(* CODESYS project SNDLTN_Domoticz.library
   Company: Sandolution
   Title: SNDLTN_Domoticz
   Description: Library to control Domoticz from a CoDeSys PLC using JSON over HTTP/MQTT.
   Author: S. Verbeek
   Version: 2.5.201026

Project tree, tasks and I/O mapping:
  libraries: StringUtils, * (System); Standard, * (System); CAA Real Time Clock Extern, * (CAA Technical Workgroup); SNDLTN_HTTP, 1.2.200929 (Sandolution); SNDLTN_MQTT, 1.2.200929 (Sandolution); SNDLTN_JSON, 1.2 (Sandolution)
  Constants/
    global variables Domoticz_Constants
    global variables Domoticz_Properties
  Enums/
    data type Domoticz_eErrors
    data type _Domoticz_eObjectDataType
    data type _Domoticz_eDataSource
    data type _Domoticz_eCommandType
    data type Domoticz_eSValues_Colors
    data type Domoticz_eHumidityStatus
    data type Domoticz_eForecast
    data type _Domoticz_eHTTP_PropertyNames
    data type Domoticz_eSValues_TempHumBaro
    data type Domoticz_eSValues_General
    data type Domoticz_eSValues_Wind
    data type Domoticz_eSValues_Rain
    data type Domoticz_eSValues_Usage
    data type Domoticz_eSValues_P1
    data type _Domoticz_eMQTT_PropertyNames
  Function Blocks/
    Objects/
      function block _Domoticz_ObjectBool_InOut [ST]: Main
      function block _Domoticz_ObjectReal_InOut [ST]: Main, rScalingSet
      function block _Domoticz_ObjectInt_InOut [ST]: Main, xUseOnlyNValue
      function block _Domoticz_Object [ST]: Main, ForceSet, RegisterSlave, xUpdateReceived, xDataTimedOut, sDeviceType, dtLastUpdate, eDataSource, eCommandType
      function block _Domoticz_ObjectString_InOut [ST]: Main
      function block _Domoticz_ObjectArrayReal_InOut [ST]: Main, arScalingSet
      function block _Domoticz_ObjectArrayReal_Out [ST]: Main, arScalingAct
      function block _Domoticz_ObjectBool_Out [ST]: Main
      function block _Domoticz_ObjectInt_Out [ST]: Main, iValueSetLimitLow, iValueSetLimitHigh
      function block _Domoticz_ObjectReal_Out [ST]: Main, rScalingAct
      function block _Domoticz_ObjectString_Out [ST]: Main
    Hardware/
      Weather/
        function block Domoticz_DarkSky [ST]: Main
        function block Domoticz_BuienAlarm [ST]: Main
        function block Domoticz_BuienRadar [ST]: Main
        function block Domoticz_OpenWeatherMap [ST]: Main
        function block Domoticz_WeatherBit [ST]: Main
        function block Domoticz_SunMoon [ST]: Main
        function block Domoticz_AccuWeather [ST]: Main
        function block Domoticz_BuienRadar_Forecast [ST]: Main
      Custom/
        function block Domoticz_CustomDimmer [ST]: Main, xUseOnlyNValue
        function block Domoticz_CustomSwitch [ST]: Main, xInvert
        function block Domoticz_CustomSensor [ST]: Main, rScalingSet, rScalingAct
        function block Domoticz_CustomString [ST]: Main
        function block Domoticz_CustomSensors [ST]: Main, arScalingSet, arScalingAct
      System/Network/
        function block Domoticz_SystemAliveChecker [ST]: Main
        function block Domoticz_MotherboardSensors [ST]: Main, rThresholdCPUHigh, rThresholdCPUMax, rThresholdMemoryHigh, rThresholdMemoryMax, rThresholdHDDHigh, rThresholdHDDMax, rThresholdTemperatureHigh, rThresholdTemperatureMax
        function block Domoticz_UPSMonitor [ST]: Main, rThresholdChargeLevelLow, rThresholdChargeLevelCritical, rThresholdLoadLevelHigh, rThresholdLoadLevelMax, rThresholdFrequency, rThresholdVoltage
        function block Domoticz_SpeedTest [ST]: Main, tThresholdPingHigh, rThresholdDownloadSpeedLow, rThresholdUploadSpeedLow
      Devices/
        function block Domoticz_MiFlora [ST]: Main, rThresholdMoistureLow, rThresholdFertilityLow
        function block Domoticz_HueLight [ST]: Main, tFadeTime, tFadeUpdateTime, xFading
        function block Domoticz_Tasmota [ST]: Main, rThresholdCurrentHigh, rThresholdCurrentMax, rThresholdPowerUsageHigh, rThresholdPowerUsageToday, rThresholdTemperatureHigh, rThresholdTemperatureLow, rThresholdHumidityHigh, rThresholdHumidityLow, rThresholdCarbonDioxideHigh, rThresholdCarbonDioxideCritical, rThresholdParticlesHigh_1um, rThresholdParticlesHigh_2_5um, rThresholdParticlesHigh_10um, rThresholdVoltage
        function block Domoticz_GoogleDevices [ST]: Main
        function block Domoticz_Life360 [ST]: Main, xArrivedHome, xLeftHome
        function block Domoticz_HueSensor [ST]: Main
        function block Domoticz_HuePlug [ST]: Main
        function block Domoticz_HueSwitch [ST]: Main
      Climate/Energy/
        function block Domoticz_NefitEasy [ST]: Main, rThresholdPressureLow, rThresholdGasUsageToday
        function block Domoticz_UsageMeter [ST]: Main, rThresholdUsageToday, sUnit
        function block Domoticz_P1Meter [ST]: Main, rThresholdGasUsageToday, rThresholdPowerUsageHigh, rThresholdPowerUsageToday, rThresholdVoltage
    Connector/
      function block _Domoticz_Connector_Out [ST]: Main, xDataTimeOut
      function block _Domoticz_Connector_InOut [ST]: tForceSetValues, Main, xForceSetValues
      function block _Domoticz_Connector [ST]: Main, sInstanceName
      function block _Domoticz_Connector_InOut_Extended [ST]: tDataTimeOut, Main
    Server/
      function block _Domoticz_Server [ST]: Main, udiUpdateRate_HTTP, HTTP_DataTwilight, MQTT_Main, HTTP_Main, MQTT_DataObject_In, MQTT_DataObject_Out, SystemTime, tSlaveErrorResetTime, Configure_AutoSyncClock, Configure_MQTT, Configure_HTTP, Configure_Twilight, xAutoReconnect, tDataForceSetValues, udiUpdateRate_MQTT, xStartUpDone, ErrorHandling, ascActiveSlaveErrors
      function block Domoticz_Server [ST]
      function block _Domoticz_Server_HTTP_Object [ST]: Main, ResetObjectData, DataObject_In
    Other/
      function block Domoticz_ServerLog [ST]: ShiftArray, Main
      function block Domoticz_ErrorInterface [ST]: Main, sErrorInfo, tErrorDelay
      function block _Domoticz_SwitchPoint [ST]: Main
  Functions/
    function _Domoticz_StringToReal [ST]
    function _Domoticz_StringToByte [ST]
    function _Domoticz_StringExtractColor [ST]
    function _Domoticz_RoundDecimals [ST]
    function _Domoticz_EqualWithWindow [ST]
    function _Domoticz_StringExtractAfterDot [ST]
    function _Domoticz_ColorFactor [ST]
  Structs/
    data type Domoticz_scObjectData
    data type Domoticz_scTwilightData
    data type Domoticz_scColorData
    data type Domoticz_scConnector
    data type Domoticz_scError
  Variables/
  Visualizations/
  text list GlobalTextList
  program ChangeLog [ST]
*)

// Enums/Domoticz_eErrors
{attribute 'qualified_only'}
{attribute 'to_string'}
TYPE Domoticz_eErrors:
(
	NoError 								:= 0,		// No error
	                                		
	//0-99 :SERVER                 		
	ServerStarting							:= 1,		//First data refresh cycle (HTTP) active
	HTTPConnectionLost						:= 10,		//Lost connection with HTTP broker
	HTTPUpdateTimeOut						:= 11,		//Timeout on last update
	MQTTConnectionLost						:= 20,		//Lost connection with MQTT broker
	MQTTUpdateTimeOut						:= 21,		//Timeout on last update
	ErrorHandlerArrayFull					:= 30,		//Array full
	ErrorHandlerEntryNotFound				:= 31,		//Entry not found in array
                                    		
	//100-199 :OBJECTS             		
	ObjectMaxReached						:= 100, 	//Maximal amount of slaves connected
	ObjectRegistrationNotPossible			:= 101,		//Register slave not possible
	ObjectInvalidData						:= 102,		//Failed during reading of HTTP data
	ObjectDataTimeOut						:= 103,		//TimeOut of received data
	                                		
	//200-999 :HARDWARE            		
	                                		
	//200-249 :Motherboard         		
	Motherboard_CpuUsageHigh				:= 210,		//Motherboard high CPU usage (>75%)
	Motherboard_CpuUsageMax					:= 211,		//Motherboard high CPU usage (>95%)
	Motherboard_MemoryUsageHigh				:= 220,		//Motherboard high memory usage (>75%)
	Motherboard_MemoryUsageMax				:= 221,		//Motherboard high memory usage (>95%)
	Motherboard_HddUsageHigh				:= 230,		//Motherboard high HDD usage (>75%)
	Motherboard_HddUsageMax					:= 231,		//Motherboard high HDD usage (>90%)
	Motherboard_TemperatureHigh				:= 240,		//Motherboard high temperature (> C60)
	Motherboard_TemperatureMax				:= 241,		//Motherboard high temperature (> C80)
	//250-299 :Speedtest           		
	SpeedTest_PingHigh						:= 260,		//Speedtest high ping
	SpeedTest_DownloadSpeedLow				:= 270,		//Speedtest download speed low
	SpeedTest_UploadSpeedLow				:= 271,		//Speedtest upload speed low                            
	//300-349 :MiFlora             		      
	MiFlora_MoistureLow						:= 310,		//MiFlora low moisture (< 25%)
	MiFlora_FertilityLow					:= 311,		//MiFlora low fertility (< 500uS/cm)
	//350-399 :Tasmota   
	Tasmota_PowerFailure					:= 350,		//Tasmota Mains voltage lost
	Tasmota_PowerUsageToday					:= 351,		//Tasmota high power usage (today)
	Tasmota_PowerUsageHigh					:= 352,		//Tasmota high actual power usage
	Tasmota_CurrentHigh						:= 355,		//Tasmota Load level at high level
	Tasmota_CurrentMax						:= 356,		//Tasmota Load level at max level        		
	Tasmota_TemperatureHigh					:= 360,		//Tasmota temperature too high
	Tasmota_TemperatureLow					:= 361,		//Tasmota temperature too low
	Tasmota_HumidityHigh					:= 365,		//Tasmota humidity too high
	Tasmota_HumidityLow						:= 366,		//Tasmota humidity too low
	Tasmota_CarbonDioxideHigh				:= 370,		//Tasmota carbondioxide high
	Tasmota_CarbonDioxideCritical			:= 371,		//Tasmota carbondioxide critical
	Tasmota_ParticlesHigh_1um				:= 380,		//Tasmota carbondioxide high PM1
	Tasmota_ParticlesHigh_2_5um				:= 381,		//Tasmota carbondioxide high PM2.5
	Tasmota_ParticlesHigh_10um				:= 382,		//Tasmota carbondioxide high PM10
	//400-449 :NefitEasy
	Nefit_PressureLow						:= 410,		//Nefit low pressure
	Nefit_GasUsageToday						:= 420,		//Nefit high gas usage (today)
	//450-499 :UsageMeter          		
	UsageMeter_UsageToday					:= 460,		//UsageMeter high usage (today)
	//500-549 :P1 Meter            		
	P1_PowerFailure							:= 510,		//P1Meter Mains voltage lost
	P1_PowerUsageToday						:= 520,		//P1Meter high power usage (today)
	P1_PowerUsageHigh						:= 521,		//P1Meter high actual power usage
	P1_GasUsageToday						:= 530,		//P1Meter high gas usage (today)
	//550-599 :UPS                 		
	UPS_PowerFailure						:= 560,		//UPS Mains voltage lost
	UPS_ChargeLevelLow						:= 570,		//UPS Capacity at warning level (<50%)
	UPS_ChargeLevelCritical					:= 571,		//UPS Capacity at critical level (<25%)
	UPS_LoadLevelHigh						:= 580,		//UPS Load level at high level (>75%)
	UPS_LoadLevelMax						:= 581,		//UPS Load level at critical level (>95%)
	UPS_BackupTime_5Min						:= 590,		//UPS Backup time (<5 min)
	UPS_BackupTime_1Min						:= 591,		//UPS Backup time (<1 min)
	//600-649
	Life360_LeftHome						:= 600,		//Life 360 left home
	Life360_ArrivedHome						:= 601,		//Life 360 arrived home
	//650-699                       		
	//700-749                       		
	//750-799                       		
	//800-849                       		
	//850-899                       		
	//900-999 :CUSTOM              		
	//Doors/Windows
	Custom_DoorOpened						:= 910,
	Custom_DoorClosed						:= 911,
	Custom_WindowOpened						:= 915,
	Custom_WindowClosed						:= 916,
	               
	//Safety     
	Custom_AlarmArmed_Stay					:= 920,
	Custom_AlarmArmed_Away					:= 921,
	Custom_AlarmDisarmed					:= 922,            		
	Custom_MovementDetected					:= 925,	
	
	//Temperature                        		  
	Custom_TemperatureHigh					:= 930,
	Custom_TemperatureLow					:= 931,
	Custom_TemperatureOutOfRange			:= 932,
	
	//Humidity                        		  
	Custom_HumidityHigh						:= 935,
	Custom_HumidityLow						:= 936,
	Custom_HumidityOutOfRange				:= 937,
	
	//Weather
	Custom_RainExpected						:= 940,
	Custom_SnowExpected						:= 941,
	Custom_FrostExpected					:= 942,
	
	//Power                   		      
	Custom_PowerFailure						:= 950,
	Custom_PowerUsageHigh					:= 951,
	Custom_PowerUsageToday					:= 952,
	         
	//System                       		
	Custom_RetainDataInvalid				:= 960,
	
	//Network
	Custom_HostUnreachable					:= 965,
	Custom_HostUnknown						:= 966,

	//Devices                               		
	Custom_ProgramComplete					:= 970,
	Custom_Triggered						:= 971,
	Custom_Activated						:= 975,
	Custom_Active							:= 976,
	Custom_Deactivated						:= 977,
	Custom_Inactive							:= 978,
	
	//Other
	Custom_Spare0							:= 990,
	Custom_Spare1							:= 991,
	Custom_Spare2							:= 992,
	Custom_Spare3							:= 993,
	Custom_Spare4							:= 994,
	Custom_Spare5							:= 995,
	Custom_Spare6							:= 996,
	Custom_Spare7							:= 997,
	Custom_Spare8							:= 998,
	Custom_Spare9							:= 999,
	
		
	//1000-1999 :HTTP ERRORS (SEE LIBRARY SNDLTN_HTTP)
	HTTP_MissingPostValue					:= 1001, 	//Current request type needs a post value
	HTTP_ParsingError						:= 1002, 	//Error while parsing the response
	HTTP_InvalidIdentifier					:= 1003,	//Invalid identifier (probably 0)
	
	//NBS errors (ported from 6001-6099)
	HTTP_NBS_TimeOut 						:= 1100,	//Time limit exceeded
	HTTP_NBS_InvalidAddress					:= 1101,	//Address invalid
	HTTP_NBS_InvalidHandle					:= 1102,	//Handle invalid
	HTTP_NBS_InvalidPointer					:= 1103,	//Data pointer invalid
	HTTP_NBS_InvalidSize					:= 1104,	//Data size invalid
	HTTP_NBS_ReceiveUDP						:= 1105,	//Error receiving data via UDP
	HTTP_NBS_SendUDP						:= 1106,	//Error sending data via UDP
	HTTP_NBS_SentIncompleteUDP				:= 1107,	//Not all data is sent.
	HTTP_NBS_OpenUDP						:= 1108,	//Couldn't open UDP connection
	HTTP_NBS_CloseUDP						:= 1109,	//Couldn't close UDP connection
	HTTP_NBS_SendTCP						:= 1110,	//Error sending data via TCP
	HTTP_NBS_ReceiveTCP						:= 1111,	//Error receiving data via TCP
	HTTP_NBS_OpenTCP						:= 1112,	//Couldn't open TCP connection
	HTTP_NBS_ConnectTCP						:= 1113,	//Couldn't connect TCP connection
	HTTP_NBS_CloseTCP						:= 1114,	//Couldn't close TCP connection
	HTTP_NBS_ServerTCP						:= 1115,	//Server error TCP
	HTTP_NBS_WrongParameter					:= 1116,	//Wrong parameters entered
	HTTP_NBS_Unknown						:= 1117,	//Not specified
	
	
	//2000-2999 :MQTT ERRORS (SEE LIBRARY SNDLTN_MQTT)
	
	//Custom errors
	MQTT_InvalidMQTT						:= 2000,	//Invalid MQTT response
	MQTT_BufferOverflow						:= 2001,	//Overflow from method
	MQTT_ConnectionLost						:= 2002,	//Connection with server lost
                                    		
	//Broker responses              		
	MQTT_RefusedProtocolVersion				:= 2010,	//Wrong protocol version
	MQTT_RefusedIdentifier					:= 2011,	//Identifier rejected
	MQTT_RefusedUserPass					:= 2012,	//Server unavailable
	MQTT_RefusedAuthorization				:= 2013,	//Authorization failed
	MQTT_ServerUnavailable					:= 2014,	//Server not available
		
	//NBS errors (ported from 6001-6099)
	MQTT_NBS_TimeOut 						:= 2100,	//Time limit exceeded
	MQTT_NBS_InvalidAddress					:= 2101,	//Address invalid
	MQTT_NBS_InvalidHandle					:= 2102,	//Handle invalid
	MQTT_NBS_InvalidPointer					:= 2103,	//Data pointer invalid
	MQTT_NBS_InvalidSize					:= 2104,	//Data size invalid
	MQTT_NBS_ReceiveUDP						:= 2105,	//Error receiving data via UDP
	MQTT_NBS_SendUDP						:= 2106,	//Error sending data via UDP
	MQTT_NBS_SentIncompleteUDP				:= 2107,	//Not all data is sent.
	MQTT_NBS_OpenUDP						:= 2108,	//Couldn't open UDP connection
	MQTT_NBS_CloseUDP						:= 2109,	//Couldn't close UDP connection
	MQTT_NBS_SendTCP						:= 2110,	//Error sending data via TCP
	MQTT_NBS_ReceiveTCP						:= 2111,	//Error receiving data via TCP
	MQTT_NBS_OpenTCP						:= 2112,	//Couldn't open TCP connection
	MQTT_NBS_ConnectTCP						:= 2113,	//Couldn't connect TCP connection
	MQTT_NBS_CloseTCP						:= 2114,	//Couldn't close TCP connection
	MQTT_NBS_ServerTCP						:= 2115,	//Server error TCP
	MQTT_NBS_WrongParameter					:= 2116,	//Wrong parameters entered
	MQTT_NBS_Unknown						:= 2117,	//Not specified
		
	//3000-3999 :JSON ERRORS (SEE LIBRARY SNDLTN_JSON)
	JSON_PropertiesArrayToSmall 			:= 3000,	//JSON Parser output array to small
	JSON_PropertySizeToSmall 				:= 3001		//JSON Size to small
);
END_TYPE

// Enums/_Domoticz_eObjectDataType
{attribute 'qualified_only'}
{attribute 'strict'}
{attribute 'conditionalshow'}
{attribute 'to_string'}
TYPE _Domoticz_eObjectDataType :
(
	NotUsed := 0,
	Identifier,
	Name,
	nValue,
	sValue1,
	sValue2,
	sValue3,
	sValue4,
	sValue5,
	sValue6,
	Color
);
END_TYPE

// Structs/Domoticz_scObjectData
TYPE Domoticz_scObjectData :
STRUCT
	//General
	uiIdentifier	:UINT;													//Identifier
	                  
	dtLastUpdate	:DATE_AND_TIME;											//Value latest updated
	dtTimeStamp		:DATE_AND_TIME;											//Latest read update
	                  
	asValue			:ARRAY[1..Domoticz_Constants.uiMaxSValues] OF STRING(JSON_Properties.uiJSONMaxPropertySize);	//Contains value if string
	iValue			:INT;													//Contains value if number
	
	//Indicate source of data
	eSource			:_Domoticz_eDataSource;									//1=MQTT 2=HTTP
	
	//Type of command (outgoing data)
	{attribute 'conditionalshow'}
	eCommand		:_Domoticz_eCommandType;								//Type of command to send
	
	{attribute 'conditionalshow'}
	sDeviceType		:STRING(Domoticz_Constants.uiObjectData_Type);			//Type of device

END_STRUCT
END_TYPE

// Structs/Domoticz_scTwilightData
TYPE Domoticz_scTwilightData :
STRUCT
	//Time
	dtSystem				:DATE_AND_TIME;
	todSystem				:TIME_OF_DAY;	
	dtServer				:DATE_AND_TIME;			//Server time is only retreived at twilight update interval
                              
	axHours					:ARRAY[0..23] OF BOOL;
                              
	xAstronomicRise			:BOOL;
	todAstronomicRise		:TIME_OF_DAY;
	                          
	xNauticRise				:BOOL;
	todNauticRise			:TIME_OF_DAY;
		                      
	xCivilRise				:BOOL;
	todCivilRise			:TIME_OF_DAY;
	                          
	xPreSunRise				:BOOL;
	todPreSunRise			:TIME_OF_DAY;
	xSunRise				:BOOL;
	todSunRise				:TIME_OF_DAY;
	xPostSunRise			:BOOL;
	todPostSunRise			:TIME_OF_DAY;
                              
	xSunAtSouth				:BOOL;
	todSunAtSouth			:TIME_OF_DAY;
	                          
	xPreSunSet				:BOOL;
	todPreSunSet			:TIME_OF_DAY;
	xSunSet					:BOOL;
	todSunSet				:TIME_OF_DAY;
	xPostSunSet				:BOOL;
	todPostSunSet			:TIME_OF_DAY;	
	                          
	xCivilSet				:BOOL;
	todCivilSet				:TIME_OF_DAY;	
	                          
	xNauticSet				:BOOL;
	todNauticSet			:TIME_OF_DAY;	
	                          
	xAstronomicSet			:BOOL;
	todAstronomicSet		:TIME_OF_DAY;
	                          
	todDayLength			:TIME_OF_DAY;
END_STRUCT
END_TYPE

// Enums/_Domoticz_eDataSource
{attribute 'qualified_only'}
{attribute 'strict'}
{attribute 'conditionalshow'} 
{attribute 'to_string'}
TYPE _Domoticz_eDataSource :
(
	All := 0,			//Allow all data sources
	MQTT,
	HTTP,
	PLC
);
END_TYPE

// Enums/_Domoticz_eCommandType
{attribute 'qualified_only'}
{attribute 'strict'}
{attribute 'conditionalshow'}
{attribute 'to_string'}
TYPE _Domoticz_eCommandType :
(
	Default := 0,
	SwitchLight,
	SwitchScene,
	SetColor,
	SetBrightness
);
END_TYPE

// Structs/Domoticz_scColorData
TYPE Domoticz_scColorData :
STRUCT
	byBrightness	:BYTE := 255;
	byRed			:BYTE;
	byGreen			:BYTE;
	byBlue			:BYTE;
	byColdWhite		:BYTE;
	byWarmWhite		:BYTE;
END_STRUCT
END_TYPE

// Enums/Domoticz_eSValues_Colors
{attribute 'qualified_only'}
{attribute 'strict'}
{attribute 'conditionalshow'}
{attribute 'to_string'}
TYPE Domoticz_eSValues_Colors :
(
	//Same order is also used in Constants.asProperty_Colors
	Brightness := 1,
	Red,
	Green,
	Blue,
	ColdWhite,
	WarmWhite
);
END_TYPE

// Structs/Domoticz_scConnector
TYPE Domoticz_scConnector :
STRUCT
	
	//Server status
	xServerConnected		:BOOL;						//Enabled and connected over HTTP and MQTT
	
	scTwilightData			:Domoticz_scTwilightData;	//Twilight data containing pulses also
	
	//Connected slave identifiers
	{attribute 'conditionalshow'}
	auiSlaveIdentifier		:ARRAY[1..Domoticz_Properties.uiMaxConnectedSlaves] OF UINT;

	uiSlaveTotal			:UINT;
	
	//Connected slave errors
	scSlaveError			:Domoticz_scError;
	
	//Forcing parameter
	tDataForceSetValues		:TIME := T#5S;				//Force set value if act is different
	
	//Input send data
	{attribute 'conditionalshow'}
	xNewObject_Tx			:BOOL;						//New values in object data
	{attribute 'conditionalshow'}
	scObjectData_Tx			:Domoticz_scObjectData;		//Object data
	
	//Output received data
	{attribute 'conditionalshow'}
	xNewObject_Rx			:BOOL;						//New values in object data
	{attribute 'conditionalshow'}
	scObjectData_Rx			:Domoticz_scObjectData;		//Object data
		
END_STRUCT
END_TYPE

// Enums/Domoticz_eHumidityStatus
{attribute 'qualified_only'}
{attribute 'to_string'} 
TYPE Domoticz_eHumidityStatus :
(
	Normal := 0,
	Comfortable := 1,
	Dry := 2,
	Wet := 3
);
END_TYPE

// Enums/Domoticz_eForecast
{attribute 'qualified_only'}
{attribute 'to_string'} 
TYPE Domoticz_eForecast :
(
	Stable := 0,
	Sunny := 1,
	PartlyCloudy := 2,
	Cloudy := 3,
	Rain := 4,
	Unknown := 5
);
END_TYPE

// Enums/_Domoticz_eHTTP_PropertyNames
{attribute 'qualified_only'}
{attribute 'strict'}
TYPE _Domoticz_eHTTP_PropertyNames :
(
	//General
	ObjectType := 1,
	Data,
	SwitchType,
	LastUpdate,
	//Switch
	Level,
	//Temp/Hum/Baro
	Temperature,
	DewPoint,
	Humidity,
	HumidityStatus,
	Barometer,
	Forecast,
	//Wind
	Speed,
	Chill,
	Gust,
	Direction,
	//Rain
	Rain,
	RainRate,
	//RGB(W)(W)
	Color,
	//Energy
	Counter,
	CounterToday,
	CounterDelivery,
	CounterDeliveryToday,
	Usage,
	UsageDelivery
);
END_TYPE

// Enums/Domoticz_eSValues_TempHumBaro
{attribute 'qualified_only'}
{attribute 'strict'}
{attribute 'conditionalshow'}
{attribute 'to_string'}
TYPE Domoticz_eSValues_TempHumBaro :
(
	//Same order is also used in Constants.asProperty_Colors
	Temperature := 1,
	Humidity,
	HumidityStatus,
	Barometer,
	Forecast,
	DewPoint
);
END_TYPE

// Enums/Domoticz_eSValues_General
{attribute 'qualified_only'}
{attribute 'strict'}
{attribute 'conditionalshow'}
{attribute 'to_string'}
TYPE Domoticz_eSValues_General :
(
	//Same order is also used in Constants.asProperty_Colors
	General := 1
);
END_TYPE

// Enums/Domoticz_eSValues_Wind
{attribute 'qualified_only'}
{attribute 'strict'}
{attribute 'conditionalshow'}
{attribute 'to_string'}
TYPE Domoticz_eSValues_Wind :
(
	//Same order is also used in Constants.asProperty_Colors
	Bearing := 1,
	Direction,
	Speed,
	Gust,
	Temperature,
	Chill
);
END_TYPE

// Enums/Domoticz_eSValues_Rain
{attribute 'qualified_only'}
{attribute 'strict'}
{attribute 'conditionalshow'}
{attribute 'to_string'}
TYPE Domoticz_eSValues_Rain :
(
	//Same order is also used in Constants.asProperty_Colors
	Rain := 1,
	RainRate
);
END_TYPE

// Enums/Domoticz_eSValues_Usage
{attribute 'qualified_only'}
{attribute 'strict'}
{attribute 'conditionalshow'}
{attribute 'to_string'}
TYPE Domoticz_eSValues_Usage :
(
	//Same order is also used in Constants.asProperty_Colors
	Usage := 1,
	UsageCumulative,	
	UsageToday 				//Additional from HTTP, not send by MQTT
);
END_TYPE

// Enums/Domoticz_eSValues_P1
{attribute 'qualified_only'}
{attribute 'strict'}
{attribute 'conditionalshow'}
{attribute 'to_string'}
TYPE Domoticz_eSValues_P1 :
(
	//Same order is also used in Constants.asProperty_Colors
	Usage1Cumulative := 1,
	Usage2Cumulative,
	Return1Cumulative,
	Return2Cumulative,
	UsageActual,
	ReturnActual,
	UsageToday,		//Additional from HTTP, not send by MQTT
	ReturnToday		//Additional from HTTP, not send by MQTT
);
END_TYPE

// Enums/_Domoticz_eMQTT_PropertyNames
{attribute 'qualified_only'}
{attribute 'strict'}
TYPE _Domoticz_eMQTT_PropertyNames :
(
	//General
	Identifier := 1,
	ObjectType,
	SwitchType,
	NValue,
	SValue1,
	SValue2,
	SValue3,
	SValue4,
	SValue5,
	SValue6,
	ColorR,
	ColorG,
	ColorB,
	ColorCW,
	ColorWW
);
END_TYPE

// Structs/Domoticz_scError
TYPE Domoticz_scError :
STRUCT
	xError				:BOOL := FALSE;
	eErrorID			:Domoticz_eErrors := Domoticz_eErrors.NoError;
	sErrorInstance		:STRING(Domoticz_Constants.uiInstanceName) := '';		//Contains instance name
	sErrorInfo			:STRING(Domoticz_Constants.uiErrorInfoSize) := '';		//Additional error info text
	udiUniqueID			:UDINT := 0;
END_STRUCT
END_TYPE

// Constants/Domoticz_Constants
{attribute 'qualified_only'}
{attribute 'conditionalshow'}
VAR_GLOBAL CONSTANT
	
	//**************************************************************************General
	uiObjectData_Type						:UINT			:= 32;		//Size of string
	uiInstanceName							:UINT			:= 128;		//Size of string
	uiMaxSValues							:UINT 			:= 8;		//Maximal S-values received, also change Domoticz_eObjectDataType and MQTT_In and HTTP_In
	uiMaxSValueSize							:UINT			:= 128;		//Maximal size of element

	uiErrorInfoSize							:UINT			:= 254;		//Size of additional error info text
	
	//**************************************************************************Types
	sType_Lighting1							:STRING(10)		:= 'Lighting 1';
	sType_Lighting2							:STRING(10)		:= 'Lighting 2';
	sType_Lighting3							:STRING(10)		:= 'Lighting 3';
	sType_Lighting4							:STRING(10)		:= 'Lighting 4';
	sType_Lighting5							:STRING(10)		:= 'Lighting 5';
	sType_LightSwitch						:STRING(12)		:= 'Light/Switch';
	sType_Security							:STRING(8)		:= 'Security';
	sSwitchType_Selector					:STRING(8)		:= 'Selector';
	sSwitchType_SelectorSwitch				:STRING(15)		:= 'Selector Switch';
	sSwitchType_Dimmer						:STRING(6)		:= 'Dimmer';
	sType_ColorSwitch						:STRING(12)		:= 'Color Switch';
	sType_TemperatureHumidityBaro			:STRING(22)		:= 'Temp + Humidity + Baro';
	sType_TemperatureHumidity				:STRING(15)		:= 'Temp + Humidity';
	sType_TemperatureBaro					:STRING(11)		:= 'Temp + Baro';
	sType_Temperature						:STRING(4)		:= 'Temp';
	sType_Humidity							:STRING(8)		:= 'Humidity';
	sType_AirQuality						:STRING(11)		:= 'Air Quality';
	sType_Wind								:STRING(4)		:= 'Wind';
	sType_Rain								:STRING(4)		:= 'Rain';
	sType_P1SmartMeter						:STRING(14)		:= 'P1 Smart Meter';
	sType_General							:STRING(7)		:= 'General';
	sType_kWh								:STRING(3)		:= 'kWh';
	sType_Energy							:STRING(6)		:= 'Energy';
	sType_Gas								:STRING(3)		:= 'Gas';
	
	//**************************************************************************Data
	sData_On								:STRING(2)		:= 'On';
	sData_Off								:STRING(3)		:= 'Off';
	sData_Open								:STRING(4)		:= 'Open';
	sData_Closed							:STRING(6)		:= 'Closed';
	sData_Locked							:STRING(6)		:= 'Locked';
	sData_Unlocked							:STRING(8)		:= 'Unlocked';
	sData_Normal							:STRING(6)		:= 'Normal';
	sData_Panic								:STRING(5)		:= 'Panic';
	
	//**************************************************************************MQTT
	//Below is present in MQTT data    
	//sPropertyMQTT_Battery					:STRING(7)		:= 'Battery';
	//sPropertyMQTT_RSSI					:STRING(4)		:= 'RSSI';
	//sPropertyMQTT_Description				:STRING(1)		:= 'description';
	sPropertyMQTT_DType						:STRING(5)		:= 'dtype';
	//sPropertyMQTT_ID						:STRING(2)		:= 'id';
	sPropertyMQTT_idx						:STRING(3)		:= 'idx';
	//sPropertyMQTT_Name					:STRING(4)		:= 'name';
	sPropertyMQTT_NValue					:STRING(6)		:= 'nvalue';
	sPropertyMQTT_SType						:STRING(5)		:= 'stype';
	sPropertyMQTT_SValue1					:STRING(7)		:= 'svalue1';
	sPropertyMQTT_SValue2					:STRING(7)		:= 'svalue2';
	sPropertyMQTT_SValue3					:STRING(7)		:= 'svalue3';
	sPropertyMQTT_SValue4					:STRING(7)		:= 'svalue4';
	sPropertyMQTT_SValue5					:STRING(7)		:= 'svalue5';
	sPropertyMQTT_SValue6					:STRING(7)		:= 'svalue6';
	//sPropertyMQTT_Unit					:STRING(4)		:= 'unit';
	//sPropertyMQTT_Color					:STRING(5)		:= 'Color';	
	
	//Commands 
	sCommandMQTT_uDevice					:STRING(19)		:= '"command":"udevice"';
	sCommandMQTT_SwitchLight				:STRING(23)		:= '"command":"switchlight"';	
	sCommandMQTT_SwitchScene				:STRING(23)		:= '"command":"switchscene"';	
	sCommandMQTT_Color						:STRING(33)		:= '"command":"setcolbrightnessvalue"';
	sCommandMQTT_Color_Value				:STRING(8)		:= '"color":';
	sCommandMQTT_Color_Mode					:STRING(1)		:= 'm';
	sCommandMQTT_Color_Temperature			:STRING(1)		:= 't';
	//Color command is defined at asProperty_Colors
	sCommandMQTT_idx						:STRING(6)		:= '"idx":';
	sCommandMQTT_sValues					:STRING(10)		:= '"svalue":"';
	sCommandMQTT_nValue						:STRING(9)		:= '"nvalue":';
	sCommandMQTT_SwitchOn					:STRING(16)		:= '"switchcmd":"On"';
	sCommandMQTT_SwitchOff					:STRING(17)		:= '"switchcmd":"Off"';
	sCommandMQTT_SwitchLevel				:STRING(23)		:= '"switchcmd":"Set Level"';
	sCommandMQTT_Level						:STRING(8)		:= '"level":';
	sCommandMQTT_Brightness					:STRING(13)		:= '"brightness":';
	
	//**************************************************************************HTTP
	sURL_HTTP								:STRING(7)		:= 'http://';	
	sURL_Twilight							:STRING(42)		:= '/json.htm?type=command&param=getSunRiseSet';
	sURL_Object								:STRING(27)		:= '/json.htm?type=devices&rid=';
	
	//Object
	sPropertyHTTP_Data						:STRING(4)		:= 'Data';
	sPropertyHTTP_Type						:STRING(4)		:= 'Type';
	sPropertyHTTP_SwitchType				:STRING(10)		:= 'SwitchType';
	sPropertyHTTP_LastUpdate				:STRING(10)		:= 'LastUpdate';
	
	//Temp/hum/baro
	sPropertyHTTP_Barometer					:STRING(9)		:= 'Barometer';
	sPropertyHTTP_Forecast					:STRING(8)		:= 'Forecast';
	sPropertyHTTP_DewPoint					:STRING(8)		:= 'DewPoint';
	sPropertyHTTP_Humidity					:STRING(8)		:= 'Humidity';
	sPropertyHTTP_HumidityStatus			:STRING(14)		:= 'HumidityStatus';
	sPropertyHTTP_Temperature				:STRING(4)		:= 'Temp';
	
	//Wind
	sPropertyHTTP_Direction					:STRING(9)		:= 'Direction';
	sPropertyHTTP_Chill						:STRING(5)		:= 'Chill';
	sPropertyHTTP_Gust						:STRING(4)		:= 'Gust';
	sPropertyHTTP_Speed						:STRING(5)		:= 'Speed';
	
	//Rain
	sPropertyHTTP_Rain						:STRING(4)		:= 'Rain';
	sPropertyHTTP_RainRate					:STRING(8)		:= 'RainRate';
	
	//RGB(W)(W)
	sPropertyHTTP_Color						:STRING(5)		:= 'Color';
	sPropertyHTTP_Level						:STRING(5)		:= 'Level';
	
	//Energy
	sPropertyHTTP_Counter					:STRING(7)		:= 'Counter';
	sPropertyHTTP_CounterToday				:STRING(12)		:= 'CounterToday';
	sPropertyHTTP_CounterDelivery			:STRING(12)		:= 'CounterDeliv';
	sPropertyHTTP_CounterDeliveryToday		:STRING(17)		:= 'CounterDelivToday';
	sPropertyHTTP_Usage						:STRING(5)		:= 'Usage';
	sPropertyHTTP_UsageDelivery				:STRING(10)		:= 'UsageDeliv';
	
	                            		
	//Twilight data                           		
	sPropertyHTTP_AstronomicRise			:STRING(17)		:= 'AstrTwilightStart';
	sPropertyHTTP_AstronomicSet				:STRING(15)		:= 'AstrTwilightEnd';
	sPropertyHTTP_CivilRise					:STRING(16)		:= 'CivTwilightStart';
	sPropertyHTTP_CivilSet					:STRING(14)		:= 'CivTwilightEnd';
	sPropertyHTTP_NauticRise				:STRING(17)		:= 'NautTwilightStart';
	sPropertyHTTP_NauticSet					:STRING(15)		:= 'NautTwilightEnd';
	sPropertyHTTP_SunRise					:STRING(7)		:= 'Sunrise';
	sPropertyHTTP_SunSet					:STRING(6)		:= 'Sunset';             		    	
	sPropertyHTTP_DayLength					:STRING(9)		:= 'DayLength';
	sPropertyHTTP_AtSouth					:STRING(10)		:= 'SunAtSouth';                            		
	sPropertyHTTP_SystemTime				:STRING(10)		:= 'ServerTime';
	
	
	//**************************************************************************COLOR
	uiProperty_ColorArraySize				:UINT := 6;
	asProperty_Colors						:ARRAY[1..uiProperty_ColorArraySize] OF STRING(2) := ['','r','g','b','cw','ww'];		//This order is also used in the array of sValues (2-6), 1 is brightness

END_VAR

// Constants/Domoticz_Properties
{attribute 'qualified_only'}
{attribute 'strict'}
VAR_GLOBAL CONSTANT
	//**************************************************************************General
	
	uiMaxConnectedSlaves					:UINT 	:= 256;			//Max connected slaves
	uiMaxHTTPConnections					:UINT 	:= 8;			//Max simultaneously connections
	uiHTTPStartUpCycles						:UINT 	:= 2;			//Number of cycles for HTTP to cycle before server reports connected
	
	uiActiveErrors							:UINT 	:= 32;			//Array size of active errors
	
	uiInterfaceLog_MaxEntries				:UINT 	:= 32;			//Maximal entries in log
	
	//MQTT Topics of Domoticz
	sMQTT_TopicReceive						:STRING(MQTT_Properties.uiMQTTMaxTopicSize) := 'domoticz/out';		//Out topic
	sMQTT_TopicSend							:STRING(MQTT_Properties.uiMQTTMaxTopicSize) := 'domoticz/in';		//In topic
	
END_VAR

// Function Blocks/Hardware/Climate/Energy/Domoticz_NefitEasy
{attribute 'conditionalshow_all_locals'}
FUNCTION_BLOCK Domoticz_NefitEasy EXTENDS _Domoticz_Connector_InOut
VAR_INPUT
	uiIdentifier_TemperatureSetpoint	:UINT;		//Setpoint temperature
	rTemperatureSetpoint_Set			:REAL;		//Setpoint temperature
	uiIdentifier_TemperatureRoom		:UINT;		//Actual temperature
	uiIdentifier_TemperatureFlow		:UINT;		//Flow temperature
	uiIdentifier_TemperatureOutside		:UINT;		//Outside temperature
	uiIdentifier_Pressure				:UINT;		//Heating pressure
	uiIdentifier_GasUsage				:UINT;		//Gas Usage
	uiIdentifier_DisplayCode			:UINT;		//Actual display code
	uiIdentifier_BoilerState			:UINT;		//Boiler state
	uiIdentifier_HotWater				:UINT;		//Hot water available
	uiIdentifier_ClockProgram			:UINT;		//Clock program
	xClockActivate						:BOOL;		//Clock program
END_VAR                          
VAR_OUTPUT                       
	rTemperatureSetpoint_Act			:REAL;
	rTemperatureRoom					:REAL;
	rTemperatureFlow					:REAL;
	rTemperatureOutside					:REAL;
	rPressure							:REAL;
	rGasUsageToday						:REAL;
	rGasUsageTotal						:REAL;
	sDisplayCode						:STRING(Domoticz_Constants.uiMaxSValuesize);
	sBoilerState						:STRING(Domoticz_Constants.uiMaxSValuesize);
	xHotWater							:BOOL;
	xClockActive						:BOOL;		//Clock program
END_VAR                         		 
VAR	                            		 
	afb_ObjectBool_InOut				:ARRAY[1..2] OF _Domoticz_ObjectBool_InOut;
	afb_ObjectReal_Out					:ARRAY[1..4] OF _Domoticz_ObjectReal_Out;
	afb_ObjectArrayReal_Out				:ARRAY[1..1] OF _Domoticz_ObjectArrayReal_Out;
	afb_ObjectReal_InOut				:ARRAY[1..1] OF _Domoticz_ObjectReal_InOut;
	afb_ObjectString_Out				:ARRAY[1..2] OF _Domoticz_ObjectString_Out;
		                        		 
	rThresholdPressureLow_int			:REAL := 1.0;
	fbSP_PressureLow					:_Domoticz_SwitchPoint;
	fbEI_PressureLow					:Domoticz_ErrorInterface;
	                            		 
	rThresholdGasUsageToday_int			:REAL := 2.0;
	fbEI_GasUsageHigh					:Domoticz_ErrorInterface;
END_VAR

IF __ISVALIDREF(scConnector) THEN
	Main();
END_IF

ACTION Main:
{attribute 'conditionalshow'}
//Call parent function
SUPER^.Main();

//Call all functions
afb_ObjectBool_InOut[1].tDataTimeOut := T#60M;
afb_ObjectBool_InOut[1](scConnector := scConnector, 	uiIdentifier := uiIdentifier_ClockProgram, 			rxUpdateInterlock := rxUpdateInterlock_int,			xValueAct => xClockActive,			xValueSet := xClockActivate);

afb_ObjectBool_InOut[2].tDataTimeOut := T#60M;
afb_ObjectBool_InOut[2](scConnector := scConnector, 	uiIdentifier := uiIdentifier_HotWater, 				rxUpdateInterlock := rxUpdateInterlock_int,			xValueAct => xHotWater);
   
afb_ObjectReal_Out[1].tDataTimeOut := T#60M;                                                     
afb_ObjectReal_Out[1](	scConnector := scConnector, 	uiIdentifier := uiIdentifier_TemperatureRoom, 		rxUpdateInterlock := rxUpdateInterlock_int,			rValueAct => rTemperatureRoom);

afb_ObjectReal_Out[2].tDataTimeOut := T#60M;
afb_ObjectReal_Out[2](	scConnector := scConnector, 	uiIdentifier := uiIdentifier_TemperatureFlow, 		rxUpdateInterlock := rxUpdateInterlock_int,			rValueAct => rTemperatureFlow);

afb_ObjectReal_Out[3].tDataTimeOut := T#60M;
afb_ObjectReal_Out[3](	scConnector := scConnector, 	uiIdentifier := uiIdentifier_TemperatureOutside, 	rxUpdateInterlock := rxUpdateInterlock_int,			rValueAct => rTemperatureOutside);

afb_ObjectReal_Out[4].tDataTimeOut := T#60M;
afb_ObjectReal_Out[4](	scConnector := scConnector, 	uiIdentifier := uiIdentifier_Pressure, 				rxUpdateInterlock := rxUpdateInterlock_int,			rValueAct => rPressure);

afb_ObjectArrayReal_Out[1].tDataTimeOut := T#60M;
afb_ObjectArrayReal_Out[1].eDataSource := _Domoticz_eDataSource.HTTP;
afb_ObjectArrayReal_Out[1](	scConnector := scConnector, uiIdentifier := uiIdentifier_GasUsage,				rxUpdateInterlock := rxUpdateInterlock_int);

afb_ObjectReal_InOut[1].tDataTimeOut := T#60M;
afb_ObjectReal_InOut[1](scConnector := scConnector, 	uiIdentifier := uiIdentifier_TemperatureSetpoint, 	rxUpdateInterlock := rxUpdateInterlock_int,			rValueAct => rTemperatureSetpoint_Act,	rValueSet := rTemperatureSetpoint_Set);

afb_ObjectString_Out[1].tDataTimeOut := T#60M;
afb_ObjectString_Out[1].eDataSource := _Domoticz_eDataSource.HTTP;
afb_ObjectString_Out[1](scConnector := scConnector, 	uiIdentifier := uiIdentifier_DisplayCode, 			rxUpdateInterlock := rxUpdateInterlock_int,			sValueAct => sDisplayCode);

afb_ObjectString_Out[2].tDataTimeOut := T#60M;
afb_ObjectString_Out[2].eDataSource := _Domoticz_eDataSource.HTTP;
afb_ObjectString_Out[2](scConnector := scConnector, 	uiIdentifier := uiIdentifier_BoilerState, 			rxUpdateInterlock := rxUpdateInterlock_int,			sValueAct => sBoilerState);

//Outputs
rGasUsageToday := afb_ObjectArrayReal_Out[1].arValueAct[Domoticz_eSValues_P1.UsageToday];
rGasUsageTotal := afb_ObjectArrayReal_Out[1].arValueAct[Domoticz_eSValues_P1.Usage1Cumulative];

//Force update of clock program
IF xForceSetValues AND xClockActivate <> xClockActive THEN
	afb_ObjectBool_InOut[1].ForceSet(tForceSetValues_int);
END_IF
//Force update of temperature when no clock program is active and temperature is set
IF xForceSetValues AND rTemperatureSetpoint_Set <> 0 AND rTemperatureSetpoint_Set <> rTemperatureSetpoint_Act AND NOT xClockActivate THEN
	afb_ObjectReal_InOut[1].ForceSet(tForceSetValues_int);
END_IF
										
//Errors
//********************************************DATA
fbEI_DataTimeOut.sInstanceName := sInstanceName;
fbEI_DataTimeOut.tErrorDelay := T#500MS;	//Give objects TIME TO be overruled BY other updates
fbEI_DataTimeOut(
	scConnector:= scConnector,
	xError:= xDataTimeOut_int
			AND (afb_ObjectBool_InOut[1].xDataTimedOut
			OR afb_ObjectBool_InOut[2].xDataTimedOut
			OR afb_ObjectReal_Out[1].xDataTimedOut
			OR afb_ObjectReal_Out[2].xDataTimedOut
			OR afb_ObjectReal_Out[3].xDataTimedOut
			OR afb_ObjectReal_Out[4].xDataTimedOut
			OR afb_ObjectArrayReal_Out[1].xDataTimedOut
			OR afb_ObjectReal_InOut[1].xDataTimedOut
			OR afb_ObjectString_Out[1].xDataTimedOut
			OR afb_ObjectString_Out[2].xDataTimedOut),
	eErrorID:= Domoticz_eErrors.ObjectDataTimeOut
);

//********************************************PRESSURE
fbSP_PressureLow(
	xEnable:= rPressure > 0,			//Note that pressure could theoretically be zero,
	rInput:= rPressure, 
	rSwitchPoint:= rThresholdPressureLow_int, 
	rHysteresis:= 0.2, 
	xInvert:= TRUE, 
	xOut=> );
fbEI_PressureLow.sInstanceName := sInstanceName;
fbEI_PressureLow.sErrorInfo := TO_STRING(_Domoticz_RoundDecimals(rPressure,1));
fbEI_PressureLow.sErrorInfo := CONCAT(fbEI_PressureLow.sErrorInfo, ' Bar');
fbEI_PressureLow(
	scConnector:= scConnector,
	xError:= fbSP_PressureLow.xOut
			AND rThresholdPressureLow_int > 0
			AND uiIdentifier_Pressure > 0,
	eErrorID:= Domoticz_eErrors.Nefit_PressureLow
);

//********************************************USAGE
fbEI_GasUsageHigh.sInstanceName := sInstanceName;
fbEI_GasUsageHigh.sErrorInfo := TO_STRING(_Domoticz_RoundDecimals(rGasUsageToday,2));
fbEI_GasUsageHigh.sErrorInfo := CONCAT(fbEI_GasUsageHigh.sErrorInfo, ' m3');
fbEI_GasUsageHigh(
	scConnector:= scConnector,
	xError:= (rGasUsageToday > rThresholdGasUsageToday_int) 
			AND rThresholdGasUsageToday_int > 0
			AND uiIdentifier_GasUsage > 0,
	eErrorID:= Domoticz_eErrors.Nefit_GasUsageToday
);
END_ACTION

{attribute 'monitoring' := 'call'} PROPERTY rThresholdPressureLow :REAL
SET
rThresholdPressureLow_int := rThresholdPressureLow;
END_SET
GET
rThresholdPressureLow := rThresholdPressureLow_int;
END_GET
END_PROPERTY

{attribute 'monitoring' := 'call'} PROPERTY rThresholdGasUsageToday :REAL
SET
rThresholdGasUsageToday_int := rThresholdGasUsageToday;
END_SET
GET
rThresholdGasUsageToday := rThresholdGasUsageToday_int;
END_GET
END_PROPERTY

END_FUNCTION_BLOCK

// Function Blocks/Connector/_Domoticz_Connector_InOut
{attribute 'conditionalshow'}
FUNCTION_BLOCK _Domoticz_Connector_InOut EXTENDS _Domoticz_Connector_Out
VAR_IN_OUT
END_VAR
VAR_INPUT
END_VAR
VAR_OUTPUT
END_VAR
VAR
	//Forcing set values
	xInit					:BOOL;
	xForceSetValues_int		:BOOL := FALSE;
	tForceSetValues_int		:TIME := T#0MS;
END_VAR

//Main called from extended functions

{attribute 'monitoring' := 'call'} PROPERTY tForceSetValues :TIME
GET
tForceSetValues := tForceSetValues_int;
END_GET
SET
//Set to {attribute 'monitoring' := 'call'} PROPERTY
IF tForceSetValues <> T#0MS THEN
	tForceSetValues_int := tForceSetValues;
//Set to internal data
ELSE
	tForceSetValues_int := scConnector.tDataForceSetValues;
END_IF
END_SET
END_PROPERTY

ACTION Main:
//Call parent function
SUPER^.Main();

//Do init config of time
IF NOT xInit
AND scConnector.tDataForceSetValues <> T#0MS THEN
	tForceSetValues := scConnector.tDataForceSetValues;
	xInit := TRUE;	//Done
END_IF
END_ACTION

{attribute 'monitoring' := 'call'} PROPERTY xForceSetValues :BOOL
SET
xForceSetValues_int := xForceSetValues;
END_SET
GET
xForceSetValues := xForceSetValues_int;
END_GET
END_PROPERTY

END_FUNCTION_BLOCK

// Function Blocks/Connector/_Domoticz_Connector_Out
{attribute 'conditionalshow'}
FUNCTION_BLOCK _Domoticz_Connector_Out EXTENDS _Domoticz_Connector
VAR_IN_OUT
END_VAR
VAR_INPUT
END_VAR
VAR_OUTPUT
END_VAR
VAR
	//Data time out
	xDataTimeOut_int		:BOOL := FALSE;
	tDataTimeOut_int		:TIME := T#0MS;
	fbEI_DataTimeOut		:Domoticz_ErrorInterface;
	
	//Interlocking of updates in hardware modules
	xUpdateInterlock_int	:BOOL;	//Update Interlock
	rxUpdateInterlock_int	:REFERENCE TO BOOL;	//Update Interlock
END_VAR

//Main called from extended functions

ACTION Main:
//Call parent function
SUPER^.Main();

//Create ref
rxUpdateInterlock_int REF= xUpdateInterlock_int;
END_ACTION

{attribute 'monitoring' := 'call'} PROPERTY xDataTimeOut :BOOL
SET
xDataTimeOut_int := xDataTimeOut;
END_SET
GET
xDataTimeOut := xDataTimeOut_int;
END_GET
END_PROPERTY

END_FUNCTION_BLOCK

// Function Blocks/Connector/_Domoticz_Connector
{attribute 'conditionalshow_all_locals'}
{attribute 'reflection'}
FUNCTION_BLOCK _Domoticz_Connector
VAR_INPUT
	scConnector				:REFERENCE TO Domoticz_scConnector;
END_VAR
VAR_OUTPUT
END_VAR
VAR
	{attribute 'instance-path'} 
	{attribute 'noinit'}
	sInstanceName_int 		:STRING(Domoticz_Constants.uiInstanceName);
END_VAR

//Main called from extended functions

ACTION Main:

END_ACTION

{attribute 'monitoring' := 'call'} PROPERTY sInstanceName :STRING(Domoticz_Constants.uiInstanceName);
SET
sInstanceName_int := sInstanceName;
END_SET
GET
sInstanceName := sInstanceName_int;
END_GET
END_PROPERTY

END_FUNCTION_BLOCK

// Function Blocks/Other/Domoticz_ErrorInterface
{attribute 'conditionalshow_all_locals'}
FUNCTION_BLOCK Domoticz_ErrorInterface EXTENDS _Domoticz_Connector
VAR_INPUT
	xError				:BOOL;
	eErrorID			:Domoticz_eErrors;
END_VAR
VAR_OUTPUT
	xBusy				:BOOL;
	xDone				:BOOL;
END_VAR
VAR
	xServerAvailable	:BOOL;
	xWaitForServer		:BOOL;
	xErrorWritten		:BOOL;
	sErrorInfo_int		:STRING(Domoticz_Constants.uiErrorInfoSize) := '';	//Additional error info text
	tErrorDelay_int		:TIME := T#1MS;	//Delay error
	TON_ErrorDelay		:TON;
	
	udiUniqueID			:UDINT;	//Unique ID received
	
	xError_mem			:BOOL := FALSE;
	sErrorInfo_mem		:STRING(Domoticz_Constants.uiErrorInfoSize);	//Additional error info text MEM
	sErrorInstance_mem	:STRING(Domoticz_Constants.uiInstanceName) := '';		//Contains instance name MEM
END_VAR

IF __ISVALIDREF(scConnector) THEN
	Main();
END_IF

ACTION Main:
{attribute 'conditionalshow'}
//Call parent function
SUPER^.Main();

//Internal status
xServerAvailable :=	scConnector.xServerConnected	//Connected
					AND NOT scConnector.scSlaveError.xError		//Connector not in use
					AND scConnector.scSlaveError.eErrorID = Domoticz_eErrors.NoError	
					AND scConnector.scSlaveError.sErrorInfo = ''
					AND scConnector.scSlaveError.sErrorInstance = ''
					AND scConnector.scSlaveError.udiUniqueID = 0;
					
//Call timer
TON_ErrorDelay(IN:= xError,	PT := tErrorDelay_int);

//Server available, write
IF (TON_ErrorDelay.Q OR xError_mem)	//Active or active before
AND xServerAvailable
AND NOT xWaitForServer
AND NOT xErrorWritten THEN
	//Internal status
	xWaitForServer := TRUE;
	xErrorWritten := FALSE;
	//Pass info for adding
	scConnector.scSlaveError.xError := TRUE;
	scConnector.scSlaveError.eErrorID := eErrorID;
	scConnector.scSlaveError.sErrorInstance := sInstanceName_int;
	scConnector.scSlaveError.sErrorInfo := sErrorInfo_int;
	scConnector.scSlaveError.udiUniqueID := 0;
	//Copy info to mem
	xError_mem := TRUE;
	sErrorInstance_mem := sInstanceName_int;
	sErrorInfo_mem := sErrorInfo_int;
	//Outputs
	xBusy := TRUE;
	xDone := FALSE;

//Error written in server, save ID
ELSIF xError_mem
AND xWaitForServer
AND scConnector.scSlaveError.udiUniqueID <> 0
AND scConnector.scSlaveError.udiUniqueID <> udiUniqueID THEN	//Already written
	//Internal status
	xWaitForServer := FALSE;
	xErrorWritten := TRUE;
	//Save response
	udiUniqueID := scConnector.scSlaveError.udiUniqueID;
	//Outputs
	xBusy := FALSE;
	xDone := TRUE;
	
//Server is done starting and is busy processing other requests
ELSIF TON_ErrorDelay.Q
AND scConnector.scSlaveError.eErrorID <> Domoticz_eErrors.ServerStarting
AND NOT xServerAvailable THEN
	//Save
	xError_mem := TRUE;
	//Outputs
	xBusy := TRUE;
	xDone := FALSE;

//Error written, remove
ELSIF NOT TON_ErrorDelay.Q 
AND xServerAvailable
AND xErrorWritten THEN
	//Internal status
	xWaitForServer := TRUE;
	xErrorWritten := FALSE;
	//Pass info for removal
	scConnector.scSlaveError.xError := TRUE;
	scConnector.scSlaveError.eErrorID := Domoticz_eErrors.NoError;	//Indicates no error present
	scConnector.scSlaveError.sErrorInstance := sErrorInstance_mem;
	scConnector.scSlaveError.sErrorInfo := sErrorInfo_mem;
	scConnector.scSlaveError.udiUniqueID := udiUniqueID;
	//Remove mem
	xError_mem := FALSE;
	sErrorInstance_mem := '';
	sErrorInfo_mem := '';
	udiUniqueID := 0;

//Error written, remove
ELSIF NOT xError_mem
AND xWaitForServer
AND scConnector.scSlaveError.udiUniqueID = 0 THEN
	//Internal status
	xWaitForServer := FALSE;
	//Outputs
	xBusy := FALSE;
	xDone := FALSE;
END_IF
END_ACTION

PROPERTY sErrorInfo :STRING(Domoticz_Constants.uiErrorInfoSize) := '';	//Additional error info text
SET
sErrorInfo_int := sErrorInfo;
END_SET
GET
sErrorInfo := sErrorInfo_int;
END_GET
END_PROPERTY

PROPERTY tErrorDelay : TIME
SET
tErrorDelay_int := tErrorDelay;
END_SET
GET
tErrorDelay := tErrorDelay_int;
END_GET
END_PROPERTY

END_FUNCTION_BLOCK

// Function Blocks/Objects/_Domoticz_ObjectBool_InOut
{attribute 'conditionalshow'}
FUNCTION_BLOCK _Domoticz_ObjectBool_InOut EXTENDS _Domoticz_ObjectBool_Out
VAR_INPUT
	xValueSet					:BOOL;
END_VAR
VAR
END_VAR

IF __ISVALIDREF(scConnector) THEN
	Main();
END_IF

ACTION Main:
{attribute 'conditionalshow'}
//Process main function
SUPER^.Main(scConnector:=scConnector);

//Transfer data to input
iValue_In := TO_INT(xValueSet);
END_ACTION

END_FUNCTION_BLOCK

// Function Blocks/Objects/_Domoticz_ObjectBool_Out
{attribute 'conditionalshow'}
FUNCTION_BLOCK _Domoticz_ObjectBool_Out EXTENDS _Domoticz_Object
VAR_OUTPUT
	xValueAct					:BOOL;
END_VAR
VAR
END_VAR

IF __ISVALIDREF(scConnector) THEN
	Main();
END_IF

ACTION Main:
{attribute 'conditionalshow'}
//Process main function
SUPER^.Main(scConnector:=scConnector);

//Transfer data to output
IF uiIdentifier_int > 0 AND xUpdateReceived_int THEN
	IF iValue_Out = 0 THEN
		xValueAct := FALSE;
	ELSIF iValue_Out >= 1 THEN
		xValueAct := TRUE;
	END_IF	
ELSIF uiIdentifier_int = 0 THEN 
	xValueAct := FALSE; 
END_IF
END_ACTION

END_FUNCTION_BLOCK

// Function Blocks/Objects/_Domoticz_Object
{attribute 'conditionalshow'}
FUNCTION_BLOCK _Domoticz_Object EXTENDS _Domoticz_Connector_InOut_Extended
VAR_INPUT
	uiIdentifier			:UINT;
	rxUpdateInterlock		:REFERENCE TO BOOL;
END_VAR                 	
VAR_OUTPUT              	
END_VAR              	
VAR	                    
	//{attribute 'instance-path'} 
	//{attribute 'noinit'}
	//Instance
	//sInstanceName 			:STRING;	

	//Store values	
	uiIdentifier_int		:UINT;	//Store identifier
	
	//Internal input data
	asValue_In				:ARRAY[1..Domoticz_Constants.uiMaxSValues] OF STRING(Domoticz_Constants.uiMaxSValuesize);	//Contains value if string
	iValue_In				:INT;
	//Data storage for change detection
	asValue_In_int			:ARRAY[1..Domoticz_Constants.uiMaxSValues] OF STRING(Domoticz_Constants.uiMaxSValuesize);	//Contains value if string
	iValue_In_int			:INT;
	
	//Internal output data
	asValue_Out				:ARRAY[1..Domoticz_Constants.uiMaxSValues] OF STRING(Domoticz_Constants.uiMaxSValuesize);	//Contains value if string
	iValue_Out				:INT;
	
	//Commands internal
	xUpdateServer			:BOOL;
	xUpdateReceived_int		:BOOL;
	xUpdateReceived_mem		:BOOL;
	xSendToServer			:BOOL := FALSE;
	
	//Other
	TON_ForceUpdate			:TON;	
	xBlockForceUpdate		:BOOL;

	eCommandTypeAct			:_Domoticz_eCommandType;//Change command type when no udevice
	eCommandTypeSet			:_Domoticz_eCommandType;//Change command type when no udevice
	
	eDataSourceFilter		:_Domoticz_eDataSource := _Domoticz_eDataSource.All;	//Filter on source of data
	eDataSourceAct			:_Domoticz_eDataSource := _Domoticz_eDataSource.All;	//Received source of data
	sDeviceType_int			:STRING(Domoticz_Constants.uiObjectData_Type);			//Type of device
	
	wX						:WORD;	//For-loop
	
	//Data timeout
	xDataTimedOut_int		:BOOL := FALSE;
	
	dtLastUpdate_int		:DATE_AND_TIME;	//Latest incoming update
	dtLastUpdate_mem		:DATE_AND_TIME;	//Saved incoming update
	dtLastUpdate_override	:DATE_AND_TIME;	//Override incoming update
	xLastUpdate_override	:BOOL;
	
	diLastUpdate			:DINT;
	diSystemTime			:DINT;
	diResult				:DINT;
END_VAR

//Main called from extended functions

//Call parent function
SUPER^.Main();

ACTION Main:
{attribute 'conditionalshow'}
//Call parent function
SUPER^.Main();

//Check if connected REF is valid
IF NOT __ISVALIDREF(scConnector) THEN
	RETURN;
END_IF

//Don't execute actions if identifier not set
IF uiIdentifier = 0 THEN
	RETURN;
//Register if ID has changed
ELSIF uiIdentifier <> uiIdentifier_int THEN
	RegisterSlave(uiIdentifier_Old:= uiIdentifier_int, uiIdentifier_New:= uiIdentifier);
	uiIdentifier_int := uiIdentifier;
END_IF

//*******************************************************************************INPUT = OUTGOING DATA = INCOMING OF SERVER

//Command is 1 cycle only
xUpdateReceived_int := FALSE;

//Delay startup of function to prevent triggering on false values
IF NOT scConnector.xServerConnected THEN
	
	//Save values at startup to prevent triggering
	//sValues
	FOR wX := 1 TO Domoticz_Constants.uiMaxSValues DO
		asValue_In_int[wX] := asValue_In[wX];
	END_FOR
	//nValue
	iValue_In_int := iValue_In;

//Check if connected and initialized
ELSIF scConnector.xServerConnected THEN
	
	//Check if data needs to be send to server
	IF NOT xSendToServer THEN
		//Check array of string
		FOR wX := 1 TO Domoticz_Constants.uiMaxSValues DO
			IF asValue_In[wX] <> asValue_In_int[wX] THEN
				xSendToServer := TRUE;
				asValue_In_int[wX] := asValue_In[wX];
			END_IF
		END_FOR
		//Check int
		IF iValue_In <> iValue_In_int THEN
			xSendToServer := TRUE;
			iValue_In_int := iValue_In;
		END_IF
		//Forced update
		IF xUpdateServer THEN
			TON_ForceUpdate(IN:=FALSE);//Call timer with false values
			xUpdateServer := FALSE;	//Reset input
			xSendToServer := TRUE;
		END_IF
		
		//Check if data is to be send > block force method and reset double sending of server udpate
		IF xSendToServer THEN
			xBlockForceUpdate := TRUE;
		END_IF
	END_IF
	
	//Server not busy > Send data
	IF xSendToServer
	AND NOT scConnector.xNewObject_Tx THEN
		//Transfer values to server
		scConnector.scObjectData_Tx.uiIdentifier := uiIdentifier_int;
		FOR wX := 1 TO Domoticz_Constants.uiMaxSValues DO
			scConnector.scObjectData_Tx.asValue[wX] := asValue_In_int[wX];
		END_FOR
		scConnector.scObjectData_Tx.iValue := iValue_In_int;
		scConnector.scObjectData_Tx.eCommand := eCommandTypeSet;
		scConnector.scObjectData_Tx.dtTimeStamp := scConnector.scTwilightData.dtSystem;
		scConnector.xNewObject_Tx := TRUE;		//Command server to send
		dtLastUpdate_int := scConnector.scObjectData_Tx.dtTimeStamp;	//Save last update
		xSendToServer := FALSE;	//Command passed on
		xBlockForceUpdate := FALSE;		//Disable block of force update
	END_IF

END_IF
	
//*******************************************************************************OUTPUT = INCOMING DATA = OUTGOING OF SERVER
//Don't wait for server connected status, because server indicates if data is available.
//New data available in server
IF scConnector.xNewObject_Rx 
AND (eDataSourceFilter = _Domoticz_eDataSource.All //Any source accepted
OR (eDataSourceFilter <> _Domoticz_eDataSource.All AND scConnector.scObjectData_Rx.eSource = eDataSourceFilter))		//Only update when source matches
AND scConnector.scObjectData_Rx.uiIdentifier = uiIdentifier_int THEN

	//Information about update
	eDataSourceAct := scConnector.scObjectData_Rx.eSource;
	eCommandTypeAct := scConnector.scObjectData_Rx.eCommand;
	sDeviceType_int := scConnector.scObjectData_Rx.sDeviceType;
	dtLastUpdate_int := scConnector.scObjectData_Rx.dtLastUpdate;
	
	//Update internal mem if changed
	IF dtLastUpdate_int <> dtLastUpdate_mem THEN
		dtLastUpdate_mem := dtLastUpdate_int;
		xLastUpdate_override := FALSE;
	END_IF
	
	//Use override if active
	IF xLastUpdate_override THEN
		dtLastUpdate_int := dtLastUpdate_override;
	END_IF
	
	//Transfer data
	FOR wX := 1 TO Domoticz_Constants.uiMaxSValues DO
		asValue_Out[wX] := scConnector.scObjectData_Rx.asValue[wX];
	END_FOR
	iValue_Out := scConnector.scObjectData_Rx.iValue;
	
	xUpdateReceived_int := TRUE;	//Update lower-laying persistent vars
	
	//Check data timeout
	IF scConnector.xServerConnected	//Only check if fully started
	AND (TO_DINT(scConnector.scTwilightData.dtSystem) - TO_DINT(dtLastUpdate_int)) > TO_DINT(TO_DT(tDataTimeOut_int))
	AND ((TO_DINT(scConnector.scTwilightData.dtSystem) - TO_DINT(dtLastUpdate_int)) > 0)	//Fix when dtLastUpdate is ahead of PLC time
	AND scConnector.scTwilightData.dtSystem <> DT#1970-1-1-00:00:00 	//Valid system time
	AND dtLastUpdate_int <> DT#1970-1-1-00:00:00 						//Valid internal time
	AND tDataTimeOut_int <> T#0MS THEN									//Valid timeout 
		diLastUpdate := TO_DINT(dtLastUpdate);
		diSystemTime := TO_DINT(scConnector.scTwilightData.dtSystem);
		diResult	:= (TO_DINT(scConnector.scTwilightData.dtSystem) - TO_DINT(dtLastUpdate));
		xDataTimedOut_int := TRUE;
	ELSE
		xDataTimedOut_int := FALSE;
	END_IF
	
END_IF

//Check 
IF __ISVALIDREF(rxUpdateInterlock) THEN
	//Set > Set status, externally not active
	IF NOT rxUpdateInterlock
	AND NOT xUpdateReceived_mem
	AND xUpdateReceived_int THEN
		xUpdateReceived_mem := TRUE;
		rxUpdateInterlock := TRUE;
	//Reset > Status set, still active
	ELSIF rxUpdateInterlock
	AND xUpdateReceived_mem
	AND NOT xUpdateReceived_int THEN
		xUpdateReceived_mem := FALSE;
		rxUpdateInterlock := FALSE;
	//External override
	ELSIF rxUpdateInterlock
	AND NOT xUpdateReceived_int THEN
		dtLastUpdate_override := scConnector.scTwilightData.dtSystem;
		xLastUpdate_override := TRUE;
	END_IF
ELSE
	xUpdateReceived_mem := FALSE;
	xLastUpdate_override := FALSE;
END_IF
END_ACTION

METHOD ForceSet
VAR_INPUT
	tForceSetValues		:TIME;
END_VAR
{warning disable C0371}
//Timer
IF ADR(scConnector) <> 0 AND tForceSetValues <> T#0MS THEN
	TON_ForceUpdate(IN:=scConnector.xServerConnected AND NOT xBlockForceUpdate, PT:=tForceSetValues);
END_IF
				
//Set output
IF TON_ForceUpdate.Q THEN
	TON_ForceUpdate(IN:=FALSE);
	xUpdateServer := TRUE;
END_IF

{warning restore C0371}
END_METHOD

{attribute 'conditionalshow'}
METHOD PRIVATE RegisterSlave :BOOL
VAR_INPUT
	uiIdentifier_Old	:UINT;
	uiIdentifier_New	:UINT;
END_VAR
VAR
	uiRegisteredIndex	:UINT;
END_VAR
{warning disable C0371}
//Delete old reference from array 
IF uiIdentifier_Old <> 0 THEN	//Valid
	FOR wX := 1 TO Domoticz_Properties.uiMaxConnectedSlaves DO
		IF scConnector.auiSlaveIdentifier[wX] = uiIdentifier_Old THEN
			scConnector.auiSlaveIdentifier[wX] := 0;
		END_IF
	END_FOR
END_IF

//Check if new one doesn't exist already
IF uiIdentifier_New <> 0 THEN	//Valid
	uiRegisteredIndex := 0;
	FOR wX := 1 TO Domoticz_Properties.uiMaxConnectedSlaves DO
		IF scConnector.auiSlaveIdentifier[wX] = uiIdentifier_New THEN
			uiRegisteredIndex := wX;
			EXIT;
		END_IF
	END_FOR
END_IF

//Add slave to array if not present yet
IF uiIdentifier_New <> 0	//Valid
AND uiRegisteredIndex = 0 THEN //Value equals zero if not changed in statement above
	FOR wX := 1 TO Domoticz_Properties.uiMaxConnectedSlaves DO
		IF scConnector.auiSlaveIdentifier[wX] = 0 THEN				//Add to empty position
			scConnector.auiSlaveIdentifier[wX] := uiIdentifier;
			EXIT;
		ELSIF wX >= Domoticz_Properties.uiMaxConnectedSlaves AND NOT scConnector.scSlaveError.xError THEN	//Registration not possible
			scConnector.scSlaveError.xError := TRUE;
			scConnector.scSlaveError.eErrorID := Domoticz_eErrors.ObjectRegistrationNotPossible;
			scConnector.scSlaveError.sErrorInstance := sInstanceName_int;
		END_IF
	END_FOR
END_IF
{warning restore C0371}
END_METHOD

PROPERTY xUpdateReceived : BOOL
GET
xUpdateReceived := xUpdateReceived_int;
END_GET
END_PROPERTY

{attribute 'monitoring' := 'call'} PROPERTY xDataTimedOut :BOOL
GET
xDataTimedOut := xDataTimedOut_int;
END_GET
END_PROPERTY

{attribute 'monitoring' := 'call'} PROPERTY sDeviceType :STRING(Domoticz_Constants.uiObjectData_Type)
GET
sDeviceType := sDeviceType_int;
END_GET
END_PROPERTY

{attribute 'monitoring' := 'call'} PROPERTY dtLastUpdate :DT
GET
dtLastUpdate := dtLastUpdate_int;
END_GET
END_PROPERTY

{attribute 'monitoring' := 'call'} PROPERTY eDataSource :_Domoticz_eDataSource
SET
eDataSourceFilter := eDataSource;
END_SET
GET
eDataSource := eDataSourceAct;
END_GET
END_PROPERTY

{attribute 'monitoring' := 'call'} PROPERTY eCommandType :_Domoticz_eCommandType
SET
eCommandTypeSet := eCommandType;
END_SET
GET
eCommandType := eCommandTypeAct;
END_GET
END_PROPERTY

END_FUNCTION_BLOCK

// Function Blocks/Connector/_Domoticz_Connector_InOut_Extended
{attribute 'conditionalshow'}
FUNCTION_BLOCK _Domoticz_Connector_InOut_Extended EXTENDS _Domoticz_Connector_InOut
VAR_IN_OUT
END_VAR
VAR_INPUT
END_VAR
VAR_OUTPUT
END_VAR
VAR
END_VAR

//Main called from extended functions

{attribute 'monitoring' := 'call'} PROPERTY tDataTimeOut :TIME
SET
tDataTimeOut_int := tDataTimeOut;
END_SET
GET
tDataTimeOut := tDataTimeOut_int;
END_GET
END_PROPERTY

ACTION Main:
//Call parent function
SUPER^.Main();
END_ACTION

END_FUNCTION_BLOCK

// Function Blocks/Objects/_Domoticz_ObjectReal_Out
{attribute 'conditionalshow'}
FUNCTION_BLOCK _Domoticz_ObjectReal_Out EXTENDS _Domoticz_Object
VAR_INPUT
END_VAR
VAR_OUTPUT
	rValueAct					:REAL;
END_VAR
VAR
	rScalingAct_int				:REAL := 1;
END_VAR

IF __ISVALIDREF(scConnector) THEN
	Main();
END_IF

ACTION Main:
{attribute 'conditionalshow'}
//Process main function
SUPER^.Main(scConnector:=scConnector);

//Transfer data to output
IF uiIdentifier_int > 0 AND xUpdateReceived_int THEN
	IF asValue_Out[1] <> '' THEN //Valid
		rValueAct := _Domoticz_StringToReal(asValue_Out[1]) * rScalingAct_int;
	END_IF
ELSIF uiIdentifier_int = 0 THEN 
	rValueAct := 0.0; 
END_IF
END_ACTION

{attribute 'monitoring' := 'call'} PROPERTY rScalingAct :REAL
SET
rScalingAct_int := rScalingAct;
END_SET
GET
rScalingAct := rScalingAct_int;
END_GET
END_PROPERTY

END_FUNCTION_BLOCK

// Functions/_Domoticz_StringToReal
{attribute 'conditionalshow_all_locals'}
{attribute 'conditionalshow'}
FUNCTION _Domoticz_StringToReal :REAL
VAR_INPUT
	sData		:STRING(Domoticz_Constants.uiMaxSValuesize);	
END_VAR
VAR
	psData		:POINTER TO STRING(Domoticz_Constants.uiMaxSValuesize);
	sFind		:STRING(Domoticz_Constants.uiMaxSValuesize);	
	psFind		:POINTER TO STRING(Domoticz_Constants.uiMaxSValuesize);
	sExtract	:STRING(Domoticz_Constants.uiMaxSValuesize);	
	psExtract	:POINTER TO STRING(Domoticz_Constants.uiMaxSValuesize);	
	
	byNumber	:BYTE;
	auiFindNumber:ARRAY[0..9] OF UINT;	//Location of number
	uiFindNumber:UINT;	//Location of first number
	uiFindSpace	:UINT;	//Location of space after first number
END_VAR

IF sData <> '' THEN
	//Load pointers
	psData := ADR(sData);
	psFind := ADR(sFind);
	psExtract := ADR(sExtract);
	
	//Find positions of all possible numbers
	FOR byNumber := 0 TO 9 DO
		sFind := TO_STRING(byNumber);
		auiFindNumber[byNumber] := TO_UINT(StrFindA(psData ,psFind, 0)); 
	END_FOR
	
	//Get number which occurs first in string
	uiFindNumber := Domoticz_Constants.uiMaxSValuesize;	//Max size of string
	FOR byNumber := 0 TO 9 DO
		IF auiFindNumber[byNumber] > 0 AND auiFindNumber[byNumber] < uiFindNumber THEN
			uiFindNumber := auiFindNumber[byNumber];
		END_IF
	END_FOR
	
	//Find space after first number
	sFind := ' ';
	uiFindSpace := TO_UINT(StrFindA(psData ,psFind, uiFindNumber)); 
	
	//Check data
	IF uiFindNumber > 0 AND uiFindNumber <> Domoticz_Constants.uiMaxSValuesize AND uiFindSpace > 0 THEN
		StrMidA(psData, Domoticz_Constants.uiMaxSValuesize, TO_INT(uiFindSpace-uiFindNumber), TO_INT(uiFindNumber), psExtract, Domoticz_Constants.uiMaxSValuesize);
	ELSE
		sExtract := sData;
	END_IF
	
	//Convert
	_Domoticz_StringToReal := TO_REAL(sExtract);
	
ELSE
	_Domoticz_StringToReal := 0.0;
END_IF

END_FUNCTION

// Function Blocks/Objects/_Domoticz_ObjectArrayReal_Out
{attribute 'conditionalshow'}
FUNCTION_BLOCK _Domoticz_ObjectArrayReal_Out EXTENDS _Domoticz_Object
VAR_OUTPUT
	arValueAct					:ARRAY[1..Domoticz_Constants.uiMaxSValues] OF REAL;
END_VAR
VAR
	arScalingAct_int			:ARRAY[1..Domoticz_Constants.uiMaxSValues] OF REAL := [Domoticz_Constants.uiMaxSValues(1)];
END_VAR

IF __ISVALIDREF(scConnector) THEN
	Main();
END_IF

ACTION Main:
{attribute 'conditionalshow'}
//Process main function
SUPER^.Main(scConnector:=scConnector);

//Transfer data to output
IF uiIdentifier_int > 0 AND xUpdateReceived_int THEN 
	FOR wX := 1 TO Domoticz_Constants.uiMaxSValues DO
		IF asValue_Out[wX] <> '' THEN	//Valid
			arValueAct[wX] := _Domoticz_StringToReal(asValue_Out[wX]) * arScalingAct_int[wX];
		END_IF
	END_FOR
	
ELSIF uiIdentifier_int = 0 THEN 
	FOR wX := 1 TO Domoticz_Constants.uiMaxSValues DO
		arValueAct[wX] := 0.0;
	END_FOR
END_IF
END_ACTION

PROPERTY arScalingAct :ARRAY[1..Domoticz_Constants.uiMaxSValues] OF REAL
SET
arScalingAct_int := arScalingAct;
END_SET
GET
arScalingAct := arScalingAct_int;
END_GET
END_PROPERTY

END_FUNCTION_BLOCK

// Function Blocks/Objects/_Domoticz_ObjectReal_InOut
{attribute 'conditionalshow'}
FUNCTION_BLOCK _Domoticz_ObjectReal_InOut EXTENDS _Domoticz_ObjectReal_Out
VAR_INPUT
	rValueSet					:REAL;
END_VAR
VAR
	rScalingSet_int				:REAL := 1;
END_VAR

IF __ISVALIDREF(scConnector) THEN
	Main();
END_IF

ACTION Main:
{attribute 'conditionalshow'}
//Process main function
SUPER^.Main(scConnector:=scConnector);

//Transfer data to input
asValue_In[1] := TO_STRING(rValueSet * rScalingSet_int);
END_ACTION

{attribute 'monitoring' := 'call'} PROPERTY rScalingSet :REAL
SET
rScalingSet_int := rScalingSet;
END_SET
GET
rScalingSet := rScalingSet_int;
END_GET
END_PROPERTY

END_FUNCTION_BLOCK

// Function Blocks/Objects/_Domoticz_ObjectString_Out
{attribute 'conditionalshow'}
FUNCTION_BLOCK _Domoticz_ObjectString_Out EXTENDS _Domoticz_Object
VAR_OUTPUT
	sValueAct					:STRING(Domoticz_Constants.uiMaxSValuesize);
END_VAR
VAR
END_VAR

IF __ISVALIDREF(scConnector) THEN
	Main();
END_IF

ACTION Main:
{attribute 'conditionalshow'}
//Process main function
SUPER^.Main(scConnector:=scConnector);

//Transfer data to output
IF uiIdentifier_int > 0 AND xUpdateReceived_int THEN 
	sValueAct := asValue_Out[1];
ELSIF uiIdentifier_int = 0 THEN 
	sValueAct := ''; 
END_IF
END_ACTION

END_FUNCTION_BLOCK

// Function Blocks/Other/_Domoticz_SwitchPoint
{attribute 'conditionalshow_all_locals'}
{attribute 'conditionalshow'}
FUNCTION_BLOCK _Domoticz_SwitchPoint
VAR_INPUT
	xEnable			:BOOL := TRUE;
	rInput			:REAL;
	rSwitchPoint	:REAL;
	rHysteresis		:REAL;
	xInvert			:BOOL;		//Hysteresis added to value instead of substracted
END_VAR
VAR_OUTPUT
	xOut			:BOOL;
END_VAR
VAR
END_VAR
//Taken from HESTIA library

Main();

ACTION Main:
IF xEnable THEN
	IF NOT xInvert THEN
		IF rInput >= rSwitchPoint THEN
			xOut := TRUE;
		ELSIF rInput <= (rSwitchPoint-rHysteresis) THEN
			xOut := FALSE;
		END_IF
	ELSIF xInvert THEN
		IF rInput <= rSwitchPoint THEN
			xOut := TRUE;
		ELSIF rInput >= (rSwitchPoint+rHysteresis) THEN
			xOut := FALSE;
		END_IF
	END_IF
ELSE
	xOut := FALSE;
END_IF
END_ACTION

END_FUNCTION_BLOCK

// Functions/_Domoticz_RoundDecimals
{attribute 'conditionalshow_all_locals'}
{attribute 'conditionalshow'}
FUNCTION _Domoticz_RoundDecimals :REAL
VAR_INPUT
	rInput			:REAL;
	byDecimals		:BYTE;
END_VAR
VAR
	lnCalculation	:LINT;
	dnMultiplier	:DINT;
END_VAR

dnMultiplier := TO_DINT(EXPT(10, byDecimals));
lnCalculation := TO_LINT(rInput * TO_REAL(dnMultiplier));
_Domoticz_RoundDecimals := (TO_REAL(lnCalculation) / TO_REAL(dnMultiplier));

END_FUNCTION

// ChangeLog
PROGRAM ChangeLog
VAR
END_VAR

//Library for interfacing with Domoticz using HTTP/MQTT/JSON.
//Relies on the SNDLTN HTTP, SNDLTN_MQTT and SNDLTN JSON library to send and retrieve data to JSON interface of Domoticz.
//Domoticz can be retreived from http://www.domoticz.com/
//Provides a single function block for setting up server connection.
//Additional function blocks can be used to control and monitor a varity of sensors/hardware.

//V2.6.201026 - October 2020:
//
//HARDWARE
//Changed all hardware FB's to reflect the rxUpdateInterlock change.
//SwitchPoint now has an enable input for controlling/resetting behaviour
//
//OBJECT
//Changed xUpdateReceived interlock to rxUpdateInterlock so that lots of interlock code could be removed.
//The interlocking now uses a single boolean which is shared between all objects in hardware.
//
//ERRORINTERFACE
//Implemented additional error info in the ErrorInterface and adjusted server to handle this.
//
//SERVER
//Implemented ascActiveSlaveErrors to get all active errors on slaves.
//Improved error handling.


//V2.6.200914 - September 2020:
//
//HARDWARE
//Fixed small bug in HueLight were forcing didn't properly work.
//Added HueSwitch for HueDimmerSwitch. Compatibility with Hue Smart Button not tested.
//Finished integration of Tasmota internal errors.
//Implemented arrived/left message in Life360 and adjusted data timeout settings.
//Added 'today' info for P1Meter and UsageMeter instead of calculating this. This way, no additional persistend data is needed.
//Small bug in SwitchPoint solved.
//
//ERRORINTERFACE
//Added ErrorInfo to slave error handling (ErrorInterface) and server. With this, additional info can be provided (such as set/act).
//Also added xBusy and xDone to ErrorInterface.
//
//SERVER
//Fixed bug in MQTT/HTTP handling to set not-used values to '' instead of '0.0'.
//MQTT values of Humidity implemented without decimals.
//
//CONSTANTS
//Changed sValues from 6 to 8 so that Counter Today (+ Counter Delivery Today) can be added for P1 meters.


//V2.5.200813 - August 2020:
//
//HARDWARE
//Added Domoticz_CustomSensors which supports multiple S-values. Mainly used for TempHumBaro.
//Implemented xUpdateReceived interlock.
//Removed Sentire integration as it is obsolete an dnot used anymore.
//Extended Tasmota with all posible sensors that can be set in the settings of a module. Other sensors have te be integrated using custom sensors.
//
//OBJECT
//Interlock of update received / data timeout possible with SET accessor of xUpdateReceived.
//ArrayReal_InOut now has an input to specify how many values must be send.
//
//SERVER
//Small bugfix where error Concat wasn't resetted and thus error instance contained previous concat value.
//Improved readability of MQTT_DataObject_In and DataObject_In (ObjectValue_HTTP). All hardcoded index values have been replaced by an ENUM (Domoticz_eSValues_XXXX).
//
//CONSTANTS
//Increased uiObjectData_Type from 16 to 32 (was to small for certain types).


//V2.5.200723 - Juli 2020:
//
//HARDWARE
//Added monitoring attribute (call) to all properties
//Increased Tasmota PowerFailure error time to 10 minutes.
//Small bugfixes in HueLight were lights wouldn't come on because they were blocked by xColorValid while still off.


//V2.5.200608 - June 2020:
//
//HARDWARE
//Moved all non-essential inputs to properties to make FB's easier and smaller to use.
//
//SERVER
//Removed ServerParameters and and created properties and methods to configure server
//
//OBJECTS
//Fixed bug where setting uiIdentifier to 0 wouldn't lead to disabling function and keeping old uiIdentifier value.


//V2.4.200402 - April 2020:
//
//DOMOTICZ
//Update to version 2020.1
//
//SERVER
//Because of Domoticz commit 20462bb values are not posted back to MQTT when updated via MQTT.
//Therefore the build-in feedback loop used to check if values are taken over correctly is broken.
//Only way to know if values are correct, is by reading the HTTP values. With big systems, it takes a while to read them.
//Therefore moved the GET and processing part to _Domoticz_ObjectValue_HTTP function block.
//Depending on Domoticz_Properties.uiMaxHTTPConnections, the registered identifiers are spread across X reading functions.
//They individually request data and update the bus.
//Implemented brightness in HTTP SetColBrightnessValue post type, no need to use seperate SetBrightness anymore for brightness settings.
//
//OBJECT
//Revisioned RegisterSlave so old identifiers gets removed from the connector before new identifier is added.
//ForceSet has a first cycle to make sure that timer is run FALSE the first time.
//Implemented DoubleSendToServer feature to be able to send a second SET command to the server. 
//This is usable when connected devices don't always respond to the first command and don't have feedback (e.g. RF).
//Added xSendToServer {attribute 'monitoring' := 'call'} PROPERTY to be able to send update to server from outside of FB - only for internal use (hidden).
//
//HARDWARE
//Increased Object_DataTimeOut for GoogleDevices FB to 24h (update rate not frequent when not in use).
//Multiplied tUpdateRate for Object_DataTimeOut in Sentire FB.
//Revisioned HueLight with better way to see if act/set are equal, using ColorFactor. Seperated SetBrightness / SetColBrightnessValue method for white/color lamps.
//
//LIBRARIES
//Update to compiler 3.5.14.40
//Updated SNDLTN_HTTP to V1.2 (inserted as explicit placeholder)
//Updated SNDLTN_MQTT to V1.2 (inserted as explicit placeholder)
//Updated SNDLTN_JSON to V1.2 (inserted as explicit placeholder)


//V2.4.200312 - March 2020:
//
//HARDWARE
//Added Tasmota plug (suitable for BW-SHP6).
//Disabled PIR xObject_DataTimeOut on HueSensor - sensor will only be updated when triggered, this shouldn't cause a data timeout.
//Disabled Object_DataTimeOut for rain & snow amount and rain & sun change in BuienRadar_Forecast, because these can be the same for a couple of days/weeks in a row.
//HotWater and ClockProgram of NefitEasy disabled because they aren't used very often. Also disabled timeout for both display codes.
//Removed tObject_DataTimeOut setting from server and implemented this for each device specificaly - times are tweaked as good as possible.
//Implemented method to set tObject_DataTimeOut on custom sensors.
//Fixed bug in HueAndMilight caused by version update of Domoticz.
//Renamed HueAndMilight to Domoticz_HueLight - MiLight goes under multiple names (AppLamp/Limitless). FB still compatible.
//
//SERVER
//Added support for Electric (Instant+Counter) type in HTTP parsing.
//Improved handling for RGB(W)(W) data type
//
//OBJECT
//Fix for when dtLastUpdate is ahead of PLC time which caused a false xObject_DataTimeOut.



//V2.4.200103 - Jan 2020:
//
//HARDWARE
//Fixed bugs regarding Object_DataTimeOut
//Added HueSensor to support Philips Hue motion sensors.
//Added HuePlug to support Philips Hue plugs (based on CustomSwitch).
//Data timeout of weather providers set to 12H:
//    (Domoticz_AccuWeather, Domoticz_BuienAlarm, Domoticz_BuienRadar, Domoticz_BuienRadar_Forecast,
//     Domoticz_DarkSky, Domoticz_OpenWeatherMap, Domoticz_SunMoon, Domoticz_WeatherBit).
//Data timeout of MiFlora set to twice the update rate.
//Added P1 Meter
//
//SERVER
//Fixed publish bug, caused when connection with broker was interrupted while publishing.
//Added support for P1 meter data in HTTP parsing.
//Added PANIC and NORMAL to _Domoticz_StringToByte to support smoke detectors.
//
//TEMPLATES
//Inserted Main actions for all template actions and calls to this in all required functions.
//
//Main function of TemplateObject_InOut has init values for tForceSetValues



//V2.4.191218 - Dec 2019:
//
//HARDWARE
//Added data timeout to guard that latest update from variables does not exceed preset time.
//Removed Root/Boot HDD from MotherboardSensors, because plugin mostly only provides one.



//V2.4.191212 - Dec 2019:
//
//HARDWARE
//Added Life360 location geofencing.
//Fixed bug which caused Objects to execute ForceUpdate when value was changed, this caused double changes. Updates are now blocked when sending an update.
//Also changed required hardware types to call ForceUpdate after calling the functions.



//V2.4.191103 - Oct 2019:
//
//CONNECTOR
//Changed all connectors to references, also implemented ISVALIDREF checks for all MAIN calls.
//
//HARDWARE
//Fixed bug in HueAndMiLight were minor rounding differences caused updating endlessly.
//Fixed bug in HueAndMiLight which caused endless updates to be send for Hue White-only lights.
//
//TWILIGHT
//Removed day of week function (moved to Hestia lib).



//V2.3 - Juli 2019:
//Additional functions required for proper working.
//
//SERVER
//Added a second MQTT client which takes care of publishing, so that the original one can take care merely of subscription messages. 
//Therefore more messages can be handled and sending does not influence receiving.
//Improved handling of HTTP messages.
//Fixed bugs regarding humidity and temp variables.
//
//CONNECTOR/TWILIGHT
//Moved twilight data into the server connector so that function blocks (Nefit, UsageMeters, EnergySupply) do not need a seperate twilight connection.
//Users can still extract it, but now from the server connector struct.
//
//HARDWARE
//Code optimization for objects, InOut types now extend Out types since they shared the same code for output variables. InOut only extends with input variables. 
//Added MiFlora, UsageMeter, CustomString (supports Text).
//Fixed force values bug in HueAndMilight.



//V2.2 - April 2019:
//
//CONNECTOR
//Redesigned _Domoticz_Object**** and _Domoticz_Object_Template (now _Domoticz_Object) to use Domoticz_scServerSlaveConnector instead of the whole server function block.
//This saves a lot of reserved memory since all hardware objects have one or more objects in them, which now use a direct struct.
//Removed _Domoticz_ServerToObject by implementing it in _Domoticz_Object_Template, because there was no need for two separate function blocks.
//Hid all internal functions and tested on CoDeSys
//
//HARDWARE
//Added hardware:GoogleDevices, EnergySupply



//V2.1 - Feb 2019:
//
//SERVER
//Because MQTT only updates on changes, data would not be loaded on start.
//Implemented a registration of slaves on the server to be able to get data of slaves via HTTP cyclically.
//This way, sensors get updated with actual values even if no MQTT updates are send by Domoticz. 
//Updates are send using the same channel/output of the server.
//Added a selectable data source, where data is not processed by slave if not from the selected data source (all/MQTT/HTTP).
//Some hardware is not time-critical and is just using HTTP data, because of formatting differences between MQTT and HTTP.
//Color controls are implemented including custom command types.
//
//HARDWARE
//Added hardware:SpeedTest / UPSMonitor / AccuWeather / BuienAlarm / BuienRadar / DarkSky / OpenWeatherMap / SunMoon / WeatherBit / HueAndMilight. 



//V2.0 - Feb 2019:
//Complete redesign of the library with a server instance and connectable slaves.
//Old version was not efficient and took too much resource in the PLC.
//Multiple servers are now also supported, because a slave has a server input.
//
//MQTT
//Implementation of SNDLTN_MQTT to receive real-time updates.
//Slaves now get their data via the MQTT update channel/output of the connected server.
//Sending is also done centrally via MQTT using a send channel/input of the connected server.
//
//TWILIGHT/TIME
//Server gets other relevant information (twilight/version) using HTTP. 
//Twilight data is also send out on the twilight channel/output of the server, including real-time system date+time.
//System date/time is automatically synced with Domoticz server if needed.
//
//HARDWARE
//Hardware can easily be added or changed because of the internal objects (_Domoticz_ObjectXXXX_XXX) for different data types.
//Each object has internally an interface for the server (_Domoticz_TemplateServerSlave).
//Objects store their values in persistent data so that this is retained at power cycle. 
//This can be only output (XX_Out) as well as input and output (XX_InOut) to limit the use persistent data. 
//
//Added hardware:MotherboardSensors / NefitEasy / SystemAliveChecker / CustomSwitch / CustomSensor / CustomDimmer.



//V1.1 - Jan 2019:
//Changed some constants into properties.
//This method requires extensive resources because each sensor sets up a HTTP connection and processes JSON data.
//A few sensors will thus work, but with more than a few the PLC will be overloaded.
//Also, polling is relativly slow and sensor changes can take a while before they are processed.
//There is a desparate need for redesign!



//V1.0 - Dec 2018:
//Implementation of server, switch and custom sensor.
//Based on polling of HTTP interface and processing data in sensor.
//Tested with version Domoticz V4.9700
//Limitations:Only single-server setup possible.

END_PROGRAM

// Function Blocks/Hardware/Custom/Domoticz_CustomSensors
{attribute 'conditionalshow_all_locals'}
FUNCTION_BLOCK Domoticz_CustomSensors EXTENDS _Domoticz_Connector_InOut_Extended
VAR_INPUT
	uiIdentifier				:UINT;	//Device to control
	arValueSet					:ARRAY[1..Domoticz_Constants.uiMaxSValues] OF REAL;		//TempHumBaro:Temperature, Humidity, Humidity_Status, Barometer, Barometer_Forecast
	uiValuesUsed				:UINT := Domoticz_Constants.uiMaxSValues;	//Amount of sValues to send
END_VAR
VAR_OUTPUT
	arValueAct					:ARRAY[1..Domoticz_Constants.uiMaxSValues] OF REAL;
END_VAR
VAR
	afb_ObjectArrayReal_InOut	:ARRAY[1..1] OF _Domoticz_ObjectArrayReal_InOut;
	arSet,arAct					:ARRAY[1..Domoticz_Constants.uiMaxSValues] OF REAL; //Calculate set/act value with scaling for forcing
	arScalingSet_int			:ARRAY[1..Domoticz_Constants.uiMaxSValues] OF REAL := [Domoticz_Constants.uiMaxSValues(1)];
	arScalingAct_int			:ARRAY[1..Domoticz_Constants.uiMaxSValues] OF REAL := [Domoticz_Constants.uiMaxSValues(1)];
	wX							:WORD;
END_VAR

IF __ISVALIDREF(scConnector) THEN
	Main();
END_IF

ACTION Main:
{attribute 'conditionalshow'}
//Call parent function
SUPER^.Main();

//Limit input value
IF uiValuesUsed < 1
OR uiValuesUsed > Domoticz_Constants.uiMaxSValues THEN
	uiValuesUsed := Domoticz_Constants.uiMaxSValues;
END_IF

//Filter set value, filter on two decimals
FOR wX := 1 TO Domoticz_Constants.uiMaxSValues DO
	arSet[wX] := _Domoticz_RoundDecimals((arValueSet[wX]*arScalingSet_int[wX]),2);	//Don't use scaling of object because of decimals
END_FOR
	
//Call all functions
afb_ObjectArrayReal_InOut[1].tDataTimeOut := tDataTimeOut_int;
afb_ObjectArrayReal_InOut[1].uiValuesUsed := uiValuesUsed;
afb_ObjectArrayReal_InOut[1](scConnector := scConnector, 	uiIdentifier := uiIdentifier,		arValueSet := arSet,		arValueAct => arAct);
		
//Filter act value, filter on two deciamls				
FOR wX := 1 TO Domoticz_Constants.uiMaxSValues DO
	arValueAct[wX] := _Domoticz_RoundDecimals((arAct[wX]*arScalingAct_int[wX]),2);	//Don't use scaling of object because of decimals
END_FOR
	
//Force status if enabled
FOR wX := 1 TO uiValuesUsed DO
	IF xForceSetValues 
	AND arSet[wX] <> arAct[wX] THEN
		afb_ObjectArrayReal_InOut[1].ForceSet(tForceSetValues_int);
	END_IF
END_FOR

//Errors
fbEI_DataTimeOut.sInstanceName := sInstanceName;
fbEI_DataTimeOut.tErrorDelay := T#500MS;	//Give objects TIME TO be overruled BY other updates
fbEI_DataTimeOut(
	scConnector:= scConnector,
	xError:= xDataTimeOut_int
			AND (afb_ObjectArrayReal_InOut[1].xDataTimedOut),
	eErrorID:= Domoticz_eErrors.ObjectDataTimeOut
);
END_ACTION

PROPERTY arScalingSet :ARRAY[1..Domoticz_Constants.uiMaxSValues] OF REAL
SET
arScalingSet_int := arScalingSet;
END_SET
GET
arScalingSet := arScalingSet_int;
END_GET
END_PROPERTY

PROPERTY arScalingAct :ARRAY[1..Domoticz_Constants.uiMaxSValues] OF REAL
SET
arScalingAct_int := arScalingAct;
END_SET
GET
arScalingAct := arScalingAct_int;
END_GET
END_PROPERTY

END_FUNCTION_BLOCK

// Function Blocks/Objects/_Domoticz_ObjectArrayReal_InOut
{attribute 'conditionalshow'}
FUNCTION_BLOCK _Domoticz_ObjectArrayReal_InOut EXTENDS _Domoticz_ObjectArrayReal_Out
VAR_INPUT
	arValueSet					:ARRAY[1..Domoticz_Constants.uiMaxSValues] OF REAL;
	uiValuesUsed				:UINT := Domoticz_Constants.uiMaxSValues;	//How many variables to send?
END_VAR
VAR
	arScalingSet_int			:ARRAY[1..Domoticz_Constants.uiMaxSValues] OF REAL := [Domoticz_Constants.uiMaxSValues(1)];
END_VAR

IF __ISVALIDREF(scConnector) THEN
	Main();
END_IF

ACTION Main:
{attribute 'conditionalshow'}
//Process main function
SUPER^.Main(scConnector:=scConnector);

//Limit input
IF uiValuesUsed < 1 THEN
	uiValuesUsed := 1;
ELSIF uiValuesUsed > Domoticz_Constants.uiMaxSValues THEN
	uiValuesUsed := Domoticz_Constants.uiMaxSValues;
END_IF

//Transfer data to input
FOR wX := 1 TO uiValuesUsed DO
	asValue_In[wX] := TO_STRING(arValueSet[wX] * arScalingSet_int[wX]);
END_FOR
IF uiValuesUsed < Domoticz_Constants.uiMaxSValues THEN
	FOR wX := (uiValuesUsed+1) TO Domoticz_Constants.uiMaxSValues DO
		asValue_In[wX] := '';
	END_FOR
END_IF
END_ACTION

PROPERTY arScalingSet :ARRAY[1..Domoticz_Constants.uiMaxSValues] OF REAL
SET
arScalingSet_int := arScalingSet;
END_SET
GET
arScalingSet := arScalingSet_int;
END_GET
END_PROPERTY

END_FUNCTION_BLOCK

// Function Blocks/Hardware/Devices/Domoticz_HueLight
{attribute 'conditionalshow_all_locals'}
FUNCTION_BLOCK Domoticz_HueLight EXTENDS _Domoticz_Connector_InOut
VAR_INPUT
	uiIdentifier				:UINT;	//Device to control
	xEnable						:BOOL;
	scColorData_Set				:Domoticz_scColorData;
END_VAR
VAR_OUTPUT
	xEnabled					:BOOL;
	scColorData_Act				:Domoticz_scColorData;
END_VAR
VAR
	xEnable_int					:BOOL;
	scColorData_Set_int			:Domoticz_scColorData;
	scColorData_Set_mem			:Domoticz_scColorData;
	byBrightness_int			:BYTE;
	sDeviceType					:STRING(Domoticz_Constants.uiObjectData_Type);			//Type of device
	rColorActSetCompare			:REAL;
	iColorActSetAmount			:INT;
	arColorActSetFactor			:ARRAY[1..Domoticz_Constants.uiProperty_ColorArraySize] OF REAL;
	xColorActValid				:BOOL;
	afb_ObjectArrayReal_InOut	:ARRAY[1..1] OF _Domoticz_ObjectArrayReal_InOut;
	
	arValueSingleStep			:ARRAY[1..Domoticz_Constants.uiProperty_ColorArraySize] OF REAL;
	tFadeTime_int				:TIME := T#1S;
	tFadeUpdateTime_int			:TIME := T#1S;
	uiFadeSteps					:UINT;
	uiFadeStepsTaken			:UINT;
	TON_Fade					:TON;
	xFading_int					:BOOL;
END_VAR

IF __ISVALIDREF(scConnector) THEN
	Main();
END_IF

ACTION Main:
{attribute 'conditionalshow'}
//Call parent function
SUPER^.Main();

//Calculate fading steps to take
IF tFadeUpdateTime_int <> T#0MS THEN
	uiFadeSteps := TO_UINT(TO_UDINT(tFadeTime)/TO_UDINT(tFadeUpdateTime_int));
END_IF

//Call all functions
afb_ObjectArrayReal_InOut[1].tDataTimeOut := T#24H;
afb_ObjectArrayReal_InOut[1](scConnector := scConnector,	uiIdentifier := uiIdentifier);

//Store devicetype internally
IF afb_ObjectArrayReal_InOut[1].sDeviceType <> sDeviceType THEN
	sDeviceType := afb_ObjectArrayReal_InOut[1].sDeviceType;
END_IF

//Set brightness value
IF xEnable 
AND ((sDeviceType = Domoticz_Constants.sType_LightSwitch 
	AND scColorData_Set.byBrightness > 0)
OR (sDeviceType = Domoticz_Constants.sType_ColorSwitch 
	AND scColorData_Set.byBrightness > 0
	AND (scColorData_Set.byRed > 0 
		OR scColorData_Set.byGreen > 0 
		OR scColorData_Set.byBlue > 0 
		OR scColorData_Set.byColdWhite > 0 
		OR scColorData_Set.byWarmWhite > 0)))
THEN

	//Use brightness to enable light
	byBrightness_int := scColorData_Set.byBrightness;
	
	IF NOT xEnable_int THEN
		//Enable mem
		xEnable_int := TRUE;
		
		//Reset color values internally
		scColorData_Set_int.byRed 			:= 0;
		scColorData_Set_int.byGreen 		:= 0;
		scColorData_Set_int.byBlue 			:= 0;
		scColorData_Set_int.byColdWhite 	:= 0;
		scColorData_Set_int.byWarmWhite 	:= 0;
		
		scColorData_Set_mem.byRed			:= 0;
		scColorData_Set_mem.byGreen			:= 0;
		scColorData_Set_mem.byBlue			:= 0;
		scColorData_Set_mem.byColdWhite 	:= 0;
		scColorData_Set_mem.byWarmWhite 	:= 0;
	END_IF
ELSE
	//Use brightness to disable light
	byBrightness_int := 0;
	
	//Disable mem
	xEnable_int := FALSE;
END_IF

//*************************************************************************************SET BRIGHTNESS & COLOR - LEVEL (HUE WHITE)
IF sDeviceType = Domoticz_Constants.sType_LightSwitch
AND NOT _Domoticz_EqualWithWindow(byBrightness_int, scColorData_Set_int.byBrightness, 1) THEN
	
	//Set mode
	afb_ObjectArrayReal_InOut[1].eCommandType := _Domoticz_eCommandType.SetBrightness;	//Don't use default uDevice
	
	//Set fading parameters
	IF uiFadeSteps > 1 THEN
		arValueSingleStep[Domoticz_eSValues_Colors.Brightness] 	:= TO_REAL(byBrightness_int)
																- TO_REAL(scColorData_Set_int.byBrightness);	//Calculate difference
		arValueSingleStep[Domoticz_eSValues_Colors.Brightness] 	:= arValueSingleStep[Domoticz_eSValues_Colors.Brightness] / uiFadeSteps;	//Divide by amount of steps
		
		xFading_int := TRUE;
		uiFadeStepsTaken := 1;
		
	ELSE
		//Transfer outgoing data
		scColorData_Set_mem.byBrightness := byBrightness_int;
	END_IF
	
	//Store data
	scColorData_Set_int.byBrightness := byBrightness_int;
	
//*************************************************************************************SET BRIGHTNESS & COLOR - COLORSWITCH
ELSIF sDeviceType = Domoticz_Constants.sType_ColorSwitch
AND (NOT _Domoticz_EqualWithWindow(byBrightness_int, scColorData_Set_int.byBrightness, 1)
OR NOT _Domoticz_EqualWithWindow(scColorData_Set.byRed, scColorData_Set_int.byRed, 1)
OR NOT _Domoticz_EqualWithWindow(scColorData_Set.byGreen, scColorData_Set_int.byGreen, 1)
OR NOT _Domoticz_EqualWithWindow(scColorData_Set.byBlue, scColorData_Set_int.byBlue, 1)
OR NOT _Domoticz_EqualWithWindow(scColorData_Set.byColdWhite, scColorData_Set_int.byColdWhite, 1)
OR NOT _Domoticz_EqualWithWindow(scColorData_Set.byWarmWhite, scColorData_Set_int.byWarmWhite, 1)) THEN
		
	//Set mode
	afb_ObjectArrayReal_InOut[1].eCommandType := _Domoticz_eCommandType.SetColor;	//Don't use default uDevice

	//Set fading parameters
	IF uiFadeSteps > 1 THEN
		arValueSingleStep[Domoticz_eSValues_Colors.Brightness] 	:= TO_REAL(byBrightness_int)
																- TO_REAL(scColorData_Set_int.byBrightness);	//Calculate difference
		arValueSingleStep[Domoticz_eSValues_Colors.Brightness] 	:= arValueSingleStep[Domoticz_eSValues_Colors.Brightness] / uiFadeSteps;	//Divide by amount of steps
		
		arValueSingleStep[Domoticz_eSValues_Colors.Red] 		:= TO_REAL(scColorData_Set.byRed)
																- TO_REAL(scColorData_Set_int.byRed);	//Calculate difference
		arValueSingleStep[Domoticz_eSValues_Colors.Red] 		:= arValueSingleStep[Domoticz_eSValues_Colors.Red] / uiFadeSteps;	//Divide by amount of steps
		
		arValueSingleStep[Domoticz_eSValues_Colors.Green] 		:= TO_REAL(scColorData_Set.byGreen)
																- TO_REAL(scColorData_Set_int.byGreen);	//Calculate difference
		arValueSingleStep[Domoticz_eSValues_Colors.Green] 		:= arValueSingleStep[Domoticz_eSValues_Colors.Green] / uiFadeSteps;	//Divide by amount of steps
		
		arValueSingleStep[Domoticz_eSValues_Colors.Blue] 		:= TO_REAL(scColorData_Set.byBlue)
																- TO_REAL(scColorData_Set_int.byBlue);	//Calculate difference
		arValueSingleStep[Domoticz_eSValues_Colors.Blue] 		:= arValueSingleStep[Domoticz_eSValues_Colors.Blue] / uiFadeSteps;	//Divide by amount of steps
		
		arValueSingleStep[Domoticz_eSValues_Colors.ColdWhite] 	:= TO_REAL(scColorData_Set.byColdWhite)
																- TO_REAL(scColorData_Set_int.byColdWhite);	//Calculate difference
		arValueSingleStep[Domoticz_eSValues_Colors.ColdWhite] 	:= arValueSingleStep[Domoticz_eSValues_Colors.ColdWhite] / uiFadeSteps;	//Divide by amount of steps
		                                                      	
		arValueSingleStep[Domoticz_eSValues_Colors.WarmWhite] 	:= TO_REAL(scColorData_Set.byWarmWhite)
																- TO_REAL(scColorData_Set_int.byWarmWhite);	//Calculate difference
		arValueSingleStep[Domoticz_eSValues_Colors.WarmWhite] 	:= arValueSingleStep[Domoticz_eSValues_Colors.WarmWhite] / uiFadeSteps;	//Divide by amount of steps

		xFading_int := TRUE;
		uiFadeStepsTaken := 1;
		
	ELSE
		//Transfer outgoing data
		scColorData_Set_mem.byBrightness	:= byBrightness_int;
		scColorData_Set_mem.byRed			:= scColorData_Set.byRed;
		scColorData_Set_mem.byGreen			:= scColorData_Set.byGreen;
		scColorData_Set_mem.byBlue			:= scColorData_Set.byBlue;
		scColorData_Set_mem.byColdWhite		:= scColorData_Set.byColdWhite;
		scColorData_Set_mem.byWarmWhite 	:= scColorData_Set.byWarmWhite;
	END_IF

	//Store data
	scColorData_Set_int.byBrightness 	:= byBrightness_int;
	scColorData_Set_int.byRed 			:= scColorData_Set.byRed;
	scColorData_Set_int.byGreen 		:= scColorData_Set.byGreen;
	scColorData_Set_int.byBlue 			:= scColorData_Set.byBlue;
	scColorData_Set_int.byColdWhite 	:= scColorData_Set.byColdWhite;
	scColorData_Set_int.byWarmWhite 	:= scColorData_Set.byWarmWhite;

	
END_IF

//*************************************************************************************FADING
//Load setpoints from fader if active
IF xFading_int THEN
	//Transfer outgoing data
	afb_ObjectArrayReal_InOut[1].arValueSet[Domoticz_eSValues_Colors.Brightness]	:= _Domoticz_RoundDecimals((((TO_REAL(scColorData_Set_mem.byBrightness)
																												+ (arValueSingleStep[Domoticz_eSValues_Colors.Brightness] * uiFadeStepsTaken)
																						)/255)*100),0);
	afb_ObjectArrayReal_InOut[1].arValueSet[Domoticz_eSValues_Colors.Red]			:= scColorData_Set_mem.byRed
																					+ (arValueSingleStep[Domoticz_eSValues_Colors.Red] * uiFadeStepsTaken);
	afb_ObjectArrayReal_InOut[1].arValueSet[Domoticz_eSValues_Colors.Green]			:= scColorData_Set_mem.byGreen
																					+ (arValueSingleStep[Domoticz_eSValues_Colors.Green] * uiFadeStepsTaken);
	afb_ObjectArrayReal_InOut[1].arValueSet[Domoticz_eSValues_Colors.Blue]			:= scColorData_Set_mem.byBlue
																					+ (arValueSingleStep[Domoticz_eSValues_Colors.Blue] * uiFadeStepsTaken);
	afb_ObjectArrayReal_InOut[1].arValueSet[Domoticz_eSValues_Colors.ColdWhite] 	:= scColorData_Set_mem.byColdWhite
																					+ (arValueSingleStep[Domoticz_eSValues_Colors.ColdWhite] * uiFadeStepsTaken);
	afb_ObjectArrayReal_InOut[1].arValueSet[Domoticz_eSValues_Colors.WarmWhite] 	:= scColorData_Set_mem.byWarmWhite
																					+ (arValueSingleStep[Domoticz_eSValues_Colors.WarmWhite] * uiFadeStepsTaken);
ELSE
	//Transfer outgoing data
	afb_ObjectArrayReal_InOut[1].arValueSet[Domoticz_eSValues_Colors.Brightness]	:= _Domoticz_RoundDecimals(((TO_REAL(scColorData_Set_mem.byBrightness)/255)*100),0);
	afb_ObjectArrayReal_InOut[1].arValueSet[Domoticz_eSValues_Colors.Red]			:= scColorData_Set_mem.byRed;
	afb_ObjectArrayReal_InOut[1].arValueSet[Domoticz_eSValues_Colors.Green]			:= scColorData_Set_mem.byGreen;
	afb_ObjectArrayReal_InOut[1].arValueSet[Domoticz_eSValues_Colors.Blue]			:= scColorData_Set_mem.byBlue;
	afb_ObjectArrayReal_InOut[1].arValueSet[Domoticz_eSValues_Colors.ColdWhite] 	:= scColorData_Set_mem.byColdWhite;
	afb_ObjectArrayReal_InOut[1].arValueSet[Domoticz_eSValues_Colors.WarmWhite] 	:= scColorData_Set_mem.byWarmWhite;
END_IF

//Increase value
IF TON_Fade.Q THEN
	IF uiFadeStepsTaken < uiFadeSteps THEN
		uiFadeStepsTaken := uiFadeStepsTaken + 1;
	ELSE
		scColorData_Set_mem := scColorData_Set_int;
		xFading_int := FALSE;
	END_IF
END_IF

//Call timer
TON_Fade(
	IN:= NOT TON_Fade.Q
		AND xFading_int,
	PT:= tFadeUpdateTime_int
);

//*************************************************************************************OUTPUTS
//Transfer incoming data
scColorData_Act.byBrightness:= TO_BYTE((afb_ObjectArrayReal_InOut[1].arValueAct[Domoticz_eSValues_Colors.Brightness]*255)/100);

xEnabled 					:= scColorData_Act.byBrightness > 0;

//Transfer output data if enabled
IF xEnabled THEN
	scColorData_Act.byRed 		:= TO_BYTE(afb_ObjectArrayReal_InOut[1].arValueAct[Domoticz_eSValues_Colors.Red]);
	scColorData_Act.byGreen 	:= TO_BYTE(afb_ObjectArrayReal_InOut[1].arValueAct[Domoticz_eSValues_Colors.Green]);
	scColorData_Act.byBlue 		:= TO_BYTE(afb_ObjectArrayReal_InOut[1].arValueAct[Domoticz_eSValues_Colors.Blue]);
	scColorData_Act.byColdWhite := TO_BYTE(afb_ObjectArrayReal_InOut[1].arValueAct[Domoticz_eSValues_Colors.ColdWhite]);
	scColorData_Act.byWarmWhite	:= TO_BYTE(afb_ObjectArrayReal_InOut[1].arValueAct[Domoticz_eSValues_Colors.WarmWhite]);
//Delete data
ELSE
	scColorData_Act.byRed 		:= 0;
	scColorData_Act.byGreen 	:= 0;
	scColorData_Act.byBlue 		:= 0;
	scColorData_Act.byColdWhite := 0;
	scColorData_Act.byWarmWhite	:= 0;
END_IF

//*************************************************************************************CHECK COLOR VALUES

IF sDeviceType = Domoticz_Constants.sType_ColorSwitch THEN
	//Check if all colors have the same scaled value
	rColorActSetCompare := 0;
	iColorActSetAmount := 0;
	
	//Red
	arColorActSetFactor[Domoticz_eSValues_Colors.Red] := _Domoticz_ColorFactor(scColorData_Act.byRed, scColorData_Set.byRed);
	//Invert value if needed
	IF arColorActSetFactor[Domoticz_eSValues_Colors.Red] > 1 THEN 
		arColorActSetFactor[Domoticz_eSValues_Colors.Red] := 1 / arColorActSetFactor[Domoticz_eSValues_Colors.Red];
	END_IF
	IF arColorActSetFactor[Domoticz_eSValues_Colors.Red] <> 0
	//AND arColorActSetFactor[Domoticz_eSValues_Colors.Red] <> -255
	AND arColorActSetFactor[Domoticz_eSValues_Colors.Red] <> 255 THEN
		IF rColorActSetCompare = 0 THEN rColorActSetCompare := arColorActSetFactor[Domoticz_eSValues_Colors.Red]; END_IF 
		iColorActSetAmount := iColorActSetAmount + 1;
	ELSE
		arColorActSetFactor[Domoticz_eSValues_Colors.Red] := 0;
	END_IF
	
	//Green
	arColorActSetFactor[Domoticz_eSValues_Colors.Green] := _Domoticz_ColorFactor(scColorData_Act.byGreen, scColorData_Set.byGreen);
	//Invert value if needed
	IF arColorActSetFactor[Domoticz_eSValues_Colors.Green] > 1 THEN 
		arColorActSetFactor[Domoticz_eSValues_Colors.Green] := 1 / arColorActSetFactor[Domoticz_eSValues_Colors.Green];
	END_IF
	IF arColorActSetFactor[Domoticz_eSValues_Colors.Green] <> 0
	//AND arColorActSetFactor[Domoticz_eSValues_Colors.Green] <> -255
	AND arColorActSetFactor[Domoticz_eSValues_Colors.Green] <> 255 THEN
		IF rColorActSetCompare = 0 THEN rColorActSetCompare := arColorActSetFactor[Domoticz_eSValues_Colors.Green]; END_IF 
		iColorActSetAmount := iColorActSetAmount + 1;
	ELSE
		arColorActSetFactor[Domoticz_eSValues_Colors.Green] := 0;
	END_IF
	
	//Blue
	arColorActSetFactor[Domoticz_eSValues_Colors.Blue] := _Domoticz_ColorFactor(scColorData_Act.byBlue, scColorData_Set.byBlue);
	//Invert value if needed
	IF arColorActSetFactor[Domoticz_eSValues_Colors.Blue] > 1 THEN 
		arColorActSetFactor[Domoticz_eSValues_Colors.Blue] := 1 / arColorActSetFactor[Domoticz_eSValues_Colors.Blue];
	END_IF
	IF arColorActSetFactor[Domoticz_eSValues_Colors.Blue] <> 0
	//AND arColorActSetFactor[Domoticz_eSValues_Colors.Blue] <> -255
	AND arColorActSetFactor[Domoticz_eSValues_Colors.Blue] <> 255 THEN
		IF rColorActSetCompare = 0 THEN rColorActSetCompare := arColorActSetFactor[Domoticz_eSValues_Colors.Blue]; END_IF 
		iColorActSetAmount := iColorActSetAmount + 1;
	ELSE
		arColorActSetFactor[Domoticz_eSValues_Colors.Blue] := 0;
	END_IF
	
	//ColdWhite
	//arColorActSetFactor[Domoticz_eSValues_Colors.ColdWhite] := _Domoticz_ColorFactor(ABS(scColorData_Act.byColdWhite - 127), ABS(scColorData_Set.byColdWhite - 127));
	arColorActSetFactor[Domoticz_eSValues_Colors.ColdWhite] := _Domoticz_ColorFactor(scColorData_Act.byColdWhite, scColorData_Set.byColdWhite);
	//Invert value if needed
	IF arColorActSetFactor[Domoticz_eSValues_Colors.ColdWhite] > 1 THEN 
		arColorActSetFactor[Domoticz_eSValues_Colors.ColdWhite] := 1 / arColorActSetFactor[Domoticz_eSValues_Colors.ColdWhite];
	END_IF
	IF arColorActSetFactor[Domoticz_eSValues_Colors.ColdWhite] <> 0
	//AND arColorActSetFactor[Domoticz_eSValues_Colors.ColdWhite] <> -255
	AND arColorActSetFactor[Domoticz_eSValues_Colors.ColdWhite] <> 255 THEN
		IF rColorActSetCompare = 0 THEN rColorActSetCompare := arColorActSetFactor[Domoticz_eSValues_Colors.ColdWhite]; END_IF 
		iColorActSetAmount := iColorActSetAmount + 1;
	ELSE
		arColorActSetFactor[Domoticz_eSValues_Colors.ColdWhite] := 0;
	END_IF
	
	//WarmWhite
	//arColorActSetFactor[Domoticz_eSValues_Colors.WarmWhite] := _Domoticz_ColorFactor(ABS(scColorData_Act.byWarmWhite - 127), ABS(scColorData_Set.byWarmWhite - 127));
	arColorActSetFactor[Domoticz_eSValues_Colors.WarmWhite] := _Domoticz_ColorFactor(scColorData_Act.byWarmWhite, scColorData_Set.byWarmWhite);
	//Invert value if needed
	IF arColorActSetFactor[Domoticz_eSValues_Colors.WarmWhite] > 1 THEN 
		arColorActSetFactor[Domoticz_eSValues_Colors.WarmWhite] := 1 / arColorActSetFactor[Domoticz_eSValues_Colors.WarmWhite];
	END_IF
	IF arColorActSetFactor[Domoticz_eSValues_Colors.WarmWhite] <> 0
	//AND arColorActSetFactor[Domoticz_eSValues_Colors.WarmWhite] <> -255
	AND arColorActSetFactor[Domoticz_eSValues_Colors.WarmWhite] <> 255 THEN
		IF rColorActSetCompare = 0 THEN rColorActSetCompare := arColorActSetFactor[Domoticz_eSValues_Colors.WarmWhite]; END_IF 
		iColorActSetAmount := iColorActSetAmount + 1;
	ELSE
		arColorActSetFactor[Domoticz_eSValues_Colors.WarmWhite] := 0;
	END_IF
	
	//Brightness
	arColorActSetFactor[Domoticz_eSValues_Colors.Brightness] := _Domoticz_ColorFactor(scColorData_Set.byBrightness, scColorData_Act.byBrightness);
	IF arColorActSetFactor[Domoticz_eSValues_Colors.Brightness] <> 0
	//AND arColorActSetFactor[Domoticz_eSValues_Colors.Brightness] <> -255
	AND arColorActSetFactor[Domoticz_eSValues_Colors.Brightness] <> 255 THEN
		IF rColorActSetCompare = 0 THEN rColorActSetCompare := arColorActSetFactor[Domoticz_eSValues_Colors.Brightness]; END_IF 
		iColorActSetAmount := iColorActSetAmount + 1;
	END_IF
	
	xColorActValid := TRUE
	AND arColorActSetFactor[Domoticz_eSValues_Colors.Brightness] < 1.1
	AND arColorActSetFactor[Domoticz_eSValues_Colors.Brightness] > 0.9
	AND ((iColorActSetAmount > 1
		AND	(_Domoticz_EqualWithWindow(rColorActSetCompare, arColorActSetFactor[Domoticz_eSValues_Colors.Red], 0.1)       OR arColorActSetFactor[Domoticz_eSValues_Colors.Red] = 0)
		AND (_Domoticz_EqualWithWindow(rColorActSetCompare, arColorActSetFactor[Domoticz_eSValues_Colors.Green], 0.1)     OR arColorActSetFactor[Domoticz_eSValues_Colors.Green] = 0)
		AND (_Domoticz_EqualWithWindow(rColorActSetCompare, arColorActSetFactor[Domoticz_eSValues_Colors.Blue], 0.1)      OR arColorActSetFactor[Domoticz_eSValues_Colors.Blue] = 0)
		AND (_Domoticz_EqualWithWindow(rColorActSetCompare, arColorActSetFactor[Domoticz_eSValues_Colors.ColdWhite], 0.1) OR arColorActSetFactor[Domoticz_eSValues_Colors.ColdWhite] = 0 OR arColorActSetFactor[Domoticz_eSValues_Colors.ColdWhite] = 1)
		AND (_Domoticz_EqualWithWindow(rColorActSetCompare, arColorActSetFactor[Domoticz_eSValues_Colors.WarmWhite], 0.1) OR arColorActSetFactor[Domoticz_eSValues_Colors.WarmWhite] = 0 OR arColorActSetFactor[Domoticz_eSValues_Colors.WarmWhite] = 1))
	OR (iColorActSetAmount = 1
		AND (_Domoticz_EqualWithWindow(rColorActSetCompare, 0, 0.1) OR _Domoticz_EqualWithWindow(rColorActSetCompare, 1, 0.1))));
		
END_IF		
	
